// TwinCAT 3 PLC project sample_delivery
// ProgramVersion: 3.1.4023.0
// libraries:
//   LCLS Sample Delivery, * (SLAC - LCLS)
//   LCLS Vacuum, * (SLAC - LCLS)
//   Tc2_Standard, * (Beckhoff Automation GmbH)
//   Tc2_System, * (Beckhoff Automation GmbH)
//   Tc3_Module, * (Beckhoff Automation GmbH)
// project tree:
//   GVLs/ GVL_RCC.TcGVL, GVL_SDS.TcGVL
//   / PlcTask.TcTTO (not stored), SerialComm.TcTTO (not stored)
//   POUs/ MAIN.TcPOU, PRG_RCC.TcPOU, SerialTxRx.TcPOU (not stored)
// real-time tasks:
//   TASK PlcTask: cycle T#10ms, priority 20, ADS port 351
//   TASK SerialComm: cycle T#5ms, priority 1, ADS port 350
// I/O:
//   DEVICE MAIN (EtherCAT), AmsNetId 0.0.0.0.2.1
//     Term 65 (EK1200)
//     Box 23 (EP9128-0021)
//     Box 31 (EP9128-0021) [EP9128-0021 8x EtherCAT junction]
//       Term 73 (EP9128-1021) [EP9128-1021 8x EtherCAT junction - Dev A]
//       Term 74 (EP9128-2021) [EP9128-2021 8x EtherCAT junction - Dev B]
//     Box 75 (EP9128-0021) [EP9128-0021 8x EtherCAT junction]
//       Term 76 (EP9128-1021) [EP9128-1021 8x EtherCAT junction - Dev A]
//       Term 77 (EP9128-2021) [EP9128-2021 8x EtherCAT junction - Dev B]
//     Box 93 (EP9128-0021) [EP9128-0021 8x EtherCAT junction]
//       FEL-SIM [EP9128-0021 8x EtherCAT junction]
//         RCC [EK1100 EtherCAT Coupler (2A E-Bus)]
//           RCC-E1 (EL2004) [EL2004 4Ch. Dig. Output 24V, 0.5A]
//           RCC-E2 (EL1004) [EL1004 4Ch. Dig. Input 24V, 3ms]
//           RCC-E3 (EL2004) [EL2004 4Ch. Dig. Output 24V, 0.5A]
//           RCC-E4 (EL2004) [EL2004 4Ch. Dig. Output 24V, 0.5A]
//           RCC-E5 (EL1004) [EL1004 4Ch. Dig. Input 24V, 3ms]
//           RCC-E6 (EL3314) [EL3314 4Ch. Ana. Input Thermocouple (TC)]
//           RCC-E7 (EL3174) [EL3174 4Ch. Ana. Input +/-10V Diff., +/-20mA SingleEnded, 16 Bit]
//           RCC-E8 (EL9011) [EL9011 End Terminal]
//         Term 87 (EP9128-1021) [EP9128-1021 8x EtherCAT junction - Dev A]
//         Term 88 (EP9128-2021) [EP9128-2021 8x EtherCAT junction - Dev B]
//       FEL-SIM-RCC (EP2339-0021) [EP2339-0021 16 Ch. Dig. Input/Output 24V, 0,5A, M8]
//       FEL-SIM-PCM (EP4374-0002) [EP4374-0002 2Ch. Ana. Input +/-10V, 0-10V, 0/4-20mA configurable; 2Ch. Ana. Output +/-10V, 0-10V, 0/4-20mA configurable]
//       Term 94 (EP9128-1021) [EP9128-1021 8x EtherCAT junction - Dev A]
//       Term 95 (EP9128-2021) [EP9128-2021 8x EtherCAT junction - Dev B]
//     WALL-RCC (EP2338-0001) [EP2338-0001 8 Ch. Dig. Input/Output 24V, 0,5A, M8]
//     WALL-RCC-PCM (EP4374-0002) [EP4374-0002 2Ch. Ana. Input +/-10V, 0-10V, 0/4-20mA configurable; 2Ch. Ana. Output +/-10V, 0-10V, 0/4-20mA configurable]
//     ALI (EP1111)
//     ALI_X (EP7041-0002)
//     ALI_Y (EP7041-0002)
//     ALI_Z (EP7041-0002)
//     ALI_X_ENC (EP5101-0011)
//     ALI_Gauges (EP3174-0002)
//     ALI_PropValve (EP7041-0002)
//     ALI_Y_ENC (EP5101-0011)
//     ALI_DIO (EP2338-0001)
//     M3 Selector A (EP1111)
//     M3 Selector A Digital IO (EP2338-1001)
//     M3 Selector A Serial IO (EP6002-0002)
//     M3 Selector B (EP1111)
//     M3 Selector B Digital IO (EP2338-1001)
//     M3 Selector B Serial IO (EP6002-0002)
//     PCM A (EP1111)
//     PCM A (EP4374-0002)
//     PCM A (EP3174-0002)
//     PCM A (EP6002-0002)
//     PCM B (EP1111)
//     PCM B (EP4374-0002)
//     PCM B (EP3174-0002)
//     PCM B (EP6002-0002)
//     Gas_Mani (EP1111)
//     Gas_Mani_NeedleValve (EP4374-0002)
//     Gas_Mani_ValveCtrl (EP2338-0001)
//     Gas_Mani_ValveRbk (EP2338-0001)
//     M3 Selector C (EP1111)
//     M3 Selector C Digital IO (EP2338-1001)
//     M3 Selector C Serial IO (EP6002-0002)
//     M3 Selector D (EP1111)
//     M3 Selector D Digital IO (EP2338-1001)
//     M3 Selector D Serial IO (EP6002-0002)
//     PCM C (EP1111)
//     PCM C (EP4374-0002)
//     PCM C (EP3174-0002)
//     PCM C (EP6002-0002)
//     PCM D (EP1111)
//     PCM D (EP4374-0002)
//     PCM D (EP3174-0002)
//     PCM D (EP6002-0002)
//     Bronkhorst MFM A
//     Bronkhorst MFM B
//     Bronkhorst MFM C
//     Bronkhorst MFM D
//     Solenoid Pair A (EP1111)
//     Solenoid Pair A Digital IO (EP2338-0001)
//     SC5 [EP9128-0021 8x EtherCAT junction]
//       Box 26 (EP9128-1021) [EP9128-1021 8x EtherCAT junction - Dev A]
//       Box 27 (EP9128-2021) [EP9128-2021 8x EtherCAT junction - Dev B]
//         SC4
//     Sensirion Flow Meter A (EP1111) [EP1111-0000 ID-Switch]
//     Sensirion Flow Meter A Serial 01 (EP6002-0002) [EP6002-0002 Interface (RS232/422/485)]
//     Sensirion Flow Meter A Serial 02 (EP6002-0002) [EP6002-0002 Interface (RS232/422/485)]
// variable links:
//   sample_delivery Instance <-> MAIN (EtherCAT)/Box 93 (EP9128-0021)/FEL-SIM-PCM (EP4374-0002)
//     PlcTask Inputs/PRG_FEL_SIM.PCM_RCC.stPropAir1.i_iPressRB <-> AI Inputs Channel 1/Value
//     PlcTask Inputs/PRG_FEL_SIM.PCM_RCC.stPropAir2.i_iPressRB <-> AI Inputs Channel 2/Value
//     PlcTask Outputs/PRG_FEL_SIM.PCM_RCC.stPropAir1.q_iPressCt <-> AO Outputs Channel 3/Analog output
//     PlcTask Outputs/PRG_FEL_SIM.PCM_RCC.stPropAir2.q_iPressCt <-> AO Outputs Channel 4/Analog output
//   sample_delivery Instance <-> MAIN (EtherCAT)/Box 93 (EP9128-0021)/FEL-SIM-RCC (EP2339-0021)
//     PlcTask Inputs/GVL_FEL_SIM.FEL_SIM_VRC_01.i_xOpnLS <-> Channel 1/Input
//     PlcTask Inputs/GVL_FEL_SIM.FEL_SIM_VRC_02.i_xOpnLS <-> Channel 2/Input
//     PlcTask Inputs/GVL_FEL_SIM.FEL_SIM_VRC_03.i_xOpnLS <-> Channel 3/Input
//     PlcTask Inputs/GVL_FEL_SIM.FEL_SIM_VRC_04.i_xOpnLS <-> Channel 4/Input
//     PlcTask Inputs/GVL_FEL_SIM.FEL_SIM_VRC_05.i_xOpnLS <-> Channel 5/Input
//     PlcTask Inputs/GVL_FEL_SIM.FEL_SIM_VRC_06.i_xOpnLS <-> Channel 6/Input
//     PlcTask Inputs/GVL_FEL_SIM.FEL_SIM_VRC_07.i_xOpnLS <-> Channel 7/Input
//     PlcTask Inputs/GVL_FEL_SIM.FEL_SIM_VRC_08.i_xOpnLS <-> Channel 8/Input
//     PlcTask Inputs/GVL_FEL_SIM.FEL_SIM_VRC_09.i_xOpnLS <-> Channel 9/Input
//     PlcTask Inputs/GVL_FEL_SIM.FEL_SIM_VRC_10.i_xOpnLS <-> Channel 10/Input
//     PlcTask Inputs/GVL_FEL_SIM.FEL_SIM_VRC_11.i_xOpnLS <-> Channel 11/Input
//     PlcTask Inputs/GVL_FEL_SIM.FEL_SIM_VRC_12.i_xOpnLS <-> Channel 12/Input
//     PlcTask Outputs/GVL_FEL_SIM.FEL_SIM_VRC_01.q_xOPN_DO <-> Channel 17/Output
//     PlcTask Outputs/GVL_FEL_SIM.FEL_SIM_VRC_02.q_xOPN_DO <-> Channel 18/Output
//     PlcTask Outputs/GVL_FEL_SIM.FEL_SIM_VRC_03.q_xOPN_DO <-> Channel 19/Output
//     PlcTask Outputs/GVL_FEL_SIM.FEL_SIM_VRC_04.q_xOPN_DO <-> Channel 20/Output
//     PlcTask Outputs/GVL_FEL_SIM.FEL_SIM_VRC_05.q_xOPN_DO <-> Channel 21/Output
//     PlcTask Outputs/GVL_FEL_SIM.FEL_SIM_VRC_06.q_xOPN_DO <-> Channel 22/Output
//     PlcTask Outputs/GVL_FEL_SIM.FEL_SIM_VRC_07.q_xOPN_DO <-> Channel 23/Output
//     PlcTask Outputs/GVL_FEL_SIM.FEL_SIM_VRC_08.q_xOPN_DO <-> Channel 24/Output
//     PlcTask Outputs/GVL_FEL_SIM.FEL_SIM_VRC_09.q_xOPN_DO <-> Channel 25/Output
//     PlcTask Outputs/GVL_FEL_SIM.FEL_SIM_VRC_10.q_xOPN_DO <-> Channel 26/Output
//     PlcTask Outputs/GVL_FEL_SIM.FEL_SIM_VRC_11.q_xOPN_DO <-> Channel 27/Output
//     PlcTask Outputs/GVL_FEL_SIM.FEL_SIM_VRC_12.q_xOPN_DO <-> Channel 28/Output
//   sample_delivery Instance <-> MAIN (EtherCAT)/Box 93 (EP9128-0021)/FEL-SIM/RCC/RCC-E6 (EL3314)
//     PlcTask Inputs/GVL_Recirculation.RCC_STC_01.bError <-> TC Inputs Channel 1/Status/Error
//     PlcTask Inputs/GVL_Recirculation.RCC_STC_01.bOverrange <-> TC Inputs Channel 1/Status/Overrange
//     PlcTask Inputs/GVL_Recirculation.RCC_STC_01.bUnderrange <-> TC Inputs Channel 1/Status/Underrange
//     PlcTask Inputs/GVL_Recirculation.RCC_STC_01.iRaw <-> TC Inputs Channel 1/Value
//   sample_delivery Instance <-> MAIN (EtherCAT)/Box 93 (EP9128-0021)/FEL-SIM/RCC/RCC-E7 (EL3174)
//     PlcTask Inputs/GVL_Recirculation.RCC_GCP_01.i_iPRESS_R <-> AI Standard Channel 1/Value
//   sample_delivery Instance <-> MAIN (EtherCAT)/Bronkhorst MFM A
//     PlcTask Inputs/GVL_SDS.BronkhorstA.stMFM.i_rFlow <-> TxPDO Map/fMeasure
//     PlcTask Outputs/GVL_SDS.BronkhorstA.stMFM.q_rSetpoint <-> RxPDO Map/fSetpoint
//   sample_delivery Instance <-> MAIN (EtherCAT)/Bronkhorst MFM B
//     PlcTask Inputs/GVL_SDS.BronkhorstB.stMFM.i_rFlow <-> TxPDO Map/fMeasure
//     PlcTask Outputs/GVL_SDS.BronkhorstB.stMFM.q_rSetpoint <-> RxPDO Map/fSetpoint
//   sample_delivery Instance <-> MAIN (EtherCAT)/Bronkhorst MFM C
//     PlcTask Inputs/GVL_SDS.BronkhorstC.stMFM.i_rFlow <-> TxPDO Map/fMeasure
//     PlcTask Outputs/GVL_SDS.BronkhorstC.stMFM.q_rSetpoint <-> RxPDO Map/fSetpoint
//   sample_delivery Instance <-> MAIN (EtherCAT)/Bronkhorst MFM D
//     PlcTask Inputs/GVL_SDS.BronkhorstD.stMFM.i_rFlow <-> TxPDO Map/fMeasure
//     PlcTask Outputs/GVL_SDS.BronkhorstD.stMFM.q_rSetpoint <-> RxPDO Map/fSetpoint
//   sample_delivery Instance <-> MAIN (EtherCAT)/Gas_Mani (EP1111)
//     PlcTask Inputs/GVL_SDS.GasMan.stBaseIO.i_SyncUnitWC <-> WcState/WcState
//   sample_delivery Instance <-> MAIN (EtherCAT)/Gas_Mani_ValveCtrl (EP2338-0001)
//     PlcTask Outputs/GVL_SDS.GasMan.stValve[{1..7}].qxDO <-> Channel {9..15}/Output  (7 links)
//   sample_delivery Instance <-> MAIN (EtherCAT)/Gas_Mani_ValveRbk (EP2338-0001)
//     PlcTask Inputs/GVL_SDS.GasMan.stValve[{1..7}].ixOPN <-> Channel {1..7}/Input  (7 links)
//   sample_delivery Instance <-> MAIN (EtherCAT)/M3 Selector A (EP1111)
//     PlcTask Inputs/GVL_SDS.M3SelectorA.stBaseIO.i_SyncUnitWC <-> WcState/WcState
//   sample_delivery Instance <-> MAIN (EtherCAT)/M3 Selector A Digital IO (EP2338-1001)
//     PlcTask Outputs/GVL_SDS.M3SelectorA.stShaker01.q_xPwrDO <-> Channel 9/Output
//     PlcTask Outputs/GVL_SDS.M3SelectorA.stShaker02.q_xPwrDO <-> Channel 10/Output
//     PlcTask Outputs/GVL_SDS.M3SelectorA.stShaker03.q_xPwrDO <-> Channel 11/Output
//     PlcTask Outputs/GVL_SDS.M3SelectorA.stShaker04.q_xPwrDO <-> Channel 12/Output
//   sample_delivery Instance <-> MAIN (EtherCAT)/M3 Selector A Serial IO (EP6002-0002)
//     SerialComm Inputs/GVL_SDS.M3SelectorA.stSensSerial.stComIn/D <-> COM TxPDO-Map Inputs Channel 1/Data In 0
//     SerialComm Inputs/GVL_SDS.M3SelectorA.stSensSerial.stComIn/D @bit {8..168 step 8} <-> COM TxPDO-Map Inputs Channel 1/Data In {1..21}  (21 links)
//     SerialComm Inputs/GVL_SDS.M3SelectorA.stSensSerial.stComIn/Status <-> COM TxPDO-Map Inputs Channel 1/Status
//     SerialComm Inputs/GVL_SDS.M3SelectorA.stViciSerial.stComIn/D <-> COM TxPDO-Map Inputs Channel 2/Data In 0
//     SerialComm Inputs/GVL_SDS.M3SelectorA.stViciSerial.stComIn/D @bit {8..168 step 8} <-> COM TxPDO-Map Inputs Channel 2/Data In {1..21}  (21 links)
//     SerialComm Inputs/GVL_SDS.M3SelectorA.stViciSerial.stComIn/Status <-> COM TxPDO-Map Inputs Channel 2/Status
//     SerialComm Outputs/GVL_SDS.M3SelectorA.stSensSerial.stComOut/Ctrl <-> COM RxPDO-Map Outputs Channel 1/Ctrl
//     SerialComm Outputs/GVL_SDS.M3SelectorA.stSensSerial.stComOut/D <-> COM RxPDO-Map Outputs Channel 1/Data Out 0
//     SerialComm Outputs/GVL_SDS.M3SelectorA.stSensSerial.stComOut/D @bit {8..168 step 8} <-> COM RxPDO-Map Outputs Channel 1/Data Out {1..21}  (21 links)
//     SerialComm Outputs/GVL_SDS.M3SelectorA.stViciSerial.stComOut/Ctrl <-> COM RxPDO-Map Outputs Channel 2/Ctrl
//     SerialComm Outputs/GVL_SDS.M3SelectorA.stViciSerial.stComOut/D <-> COM RxPDO-Map Outputs Channel 2/Data Out 0
//     SerialComm Outputs/GVL_SDS.M3SelectorA.stViciSerial.stComOut/D @bit {8..168 step 8} <-> COM RxPDO-Map Outputs Channel 2/Data Out {1..21}  (21 links)
//   sample_delivery Instance <-> MAIN (EtherCAT)/M3 Selector B (EP1111)
//     PlcTask Inputs/GVL_SDS.M3SelectorB.stBaseIO.i_SyncUnitWC <-> WcState/WcState
//   sample_delivery Instance <-> MAIN (EtherCAT)/M3 Selector B Digital IO (EP2338-1001)
//     PlcTask Outputs/GVL_SDS.M3SelectorB.stShaker01.q_xPwrDO <-> Channel 9/Output
//     PlcTask Outputs/GVL_SDS.M3SelectorB.stShaker02.q_xPwrDO <-> Channel 10/Output
//     PlcTask Outputs/GVL_SDS.M3SelectorB.stShaker03.q_xPwrDO <-> Channel 11/Output
//     PlcTask Outputs/GVL_SDS.M3SelectorB.stShaker04.q_xPwrDO <-> Channel 12/Output
//   sample_delivery Instance <-> MAIN (EtherCAT)/M3 Selector B Serial IO (EP6002-0002)
//     SerialComm Inputs/GVL_SDS.M3SelectorB.stSensSerial.stComIn/D <-> COM TxPDO-Map Inputs Channel 1/Data In 0
//     SerialComm Inputs/GVL_SDS.M3SelectorB.stSensSerial.stComIn/D @bit {8..168 step 8} <-> COM TxPDO-Map Inputs Channel 1/Data In {1..21}  (21 links)
//     SerialComm Inputs/GVL_SDS.M3SelectorB.stSensSerial.stComIn/Status <-> COM TxPDO-Map Inputs Channel 1/Status
//     SerialComm Inputs/GVL_SDS.M3SelectorB.stViciSerial.stComIn/D <-> COM TxPDO-Map Inputs Channel 2/Data In 0
//     SerialComm Inputs/GVL_SDS.M3SelectorB.stViciSerial.stComIn/D @bit {8..168 step 8} <-> COM TxPDO-Map Inputs Channel 2/Data In {1..21}  (21 links)
//     SerialComm Inputs/GVL_SDS.M3SelectorB.stViciSerial.stComIn/Status <-> COM TxPDO-Map Inputs Channel 2/Status
//     SerialComm Outputs/GVL_SDS.M3SelectorB.stSensSerial.stComOut/Ctrl <-> COM RxPDO-Map Outputs Channel 1/Ctrl
//     SerialComm Outputs/GVL_SDS.M3SelectorB.stSensSerial.stComOut/D <-> COM RxPDO-Map Outputs Channel 1/Data Out 0
//     SerialComm Outputs/GVL_SDS.M3SelectorB.stSensSerial.stComOut/D @bit {8..168 step 8} <-> COM RxPDO-Map Outputs Channel 1/Data Out {1..21}  (21 links)
//     SerialComm Outputs/GVL_SDS.M3SelectorB.stViciSerial.stComOut/Ctrl <-> COM RxPDO-Map Outputs Channel 2/Ctrl
//     SerialComm Outputs/GVL_SDS.M3SelectorB.stViciSerial.stComOut/D <-> COM RxPDO-Map Outputs Channel 2/Data Out 0
//     SerialComm Outputs/GVL_SDS.M3SelectorB.stViciSerial.stComOut/D @bit {8..168 step 8} <-> COM RxPDO-Map Outputs Channel 2/Data Out {1..21}  (21 links)
//   sample_delivery Instance <-> MAIN (EtherCAT)/M3 Selector C (EP1111)
//     PlcTask Inputs/GVL_SDS.M3SelectorC.stBaseIO.i_SyncUnitWC <-> WcState/WcState
//   sample_delivery Instance <-> MAIN (EtherCAT)/M3 Selector C Digital IO (EP2338-1001)
//     PlcTask Outputs/GVL_SDS.M3SelectorC.stShaker01.q_xPwrDO <-> Channel 9/Output
//     PlcTask Outputs/GVL_SDS.M3SelectorC.stShaker02.q_xPwrDO <-> Channel 10/Output
//     PlcTask Outputs/GVL_SDS.M3SelectorC.stShaker03.q_xPwrDO <-> Channel 11/Output
//     PlcTask Outputs/GVL_SDS.M3SelectorC.stShaker04.q_xPwrDO <-> Channel 12/Output
//   sample_delivery Instance <-> MAIN (EtherCAT)/M3 Selector C Serial IO (EP6002-0002)
//     SerialComm Inputs/GVL_SDS.M3SelectorC.stSensSerial.stComIn/D <-> COM TxPDO-Map Inputs Channel 1/Data In 0
//     SerialComm Inputs/GVL_SDS.M3SelectorC.stSensSerial.stComIn/D @bit {8..168 step 8} <-> COM TxPDO-Map Inputs Channel 1/Data In {1..21}  (21 links)
//     SerialComm Inputs/GVL_SDS.M3SelectorC.stSensSerial.stComIn/Status <-> COM TxPDO-Map Inputs Channel 1/Status
//     SerialComm Inputs/GVL_SDS.M3SelectorC.stViciSerial.stComIn/D <-> COM TxPDO-Map Inputs Channel 2/Data In 0
//     SerialComm Inputs/GVL_SDS.M3SelectorC.stViciSerial.stComIn/D @bit {8..168 step 8} <-> COM TxPDO-Map Inputs Channel 2/Data In {1..21}  (21 links)
//     SerialComm Inputs/GVL_SDS.M3SelectorC.stViciSerial.stComIn/Status <-> COM TxPDO-Map Inputs Channel 2/Status
//     SerialComm Outputs/GVL_SDS.M3SelectorC.stSensSerial.stComOut/Ctrl <-> COM RxPDO-Map Outputs Channel 1/Ctrl
//     SerialComm Outputs/GVL_SDS.M3SelectorC.stSensSerial.stComOut/D <-> COM RxPDO-Map Outputs Channel 1/Data Out 0
//     SerialComm Outputs/GVL_SDS.M3SelectorC.stSensSerial.stComOut/D @bit {8..168 step 8} <-> COM RxPDO-Map Outputs Channel 1/Data Out {1..21}  (21 links)
//     SerialComm Outputs/GVL_SDS.M3SelectorC.stViciSerial.stComOut/Ctrl <-> COM RxPDO-Map Outputs Channel 2/Ctrl
//     SerialComm Outputs/GVL_SDS.M3SelectorC.stViciSerial.stComOut/D <-> COM RxPDO-Map Outputs Channel 2/Data Out 0
//     SerialComm Outputs/GVL_SDS.M3SelectorC.stViciSerial.stComOut/D @bit {8..168 step 8} <-> COM RxPDO-Map Outputs Channel 2/Data Out {1..21}  (21 links)
//   sample_delivery Instance <-> MAIN (EtherCAT)/M3 Selector D (EP1111)
//     PlcTask Inputs/GVL_SDS.M3SelectorD.stBaseIO.i_SyncUnitWC <-> WcState/WcState
//   sample_delivery Instance <-> MAIN (EtherCAT)/M3 Selector D Digital IO (EP2338-1001)
//     PlcTask Outputs/GVL_SDS.M3SelectorD.stShaker01.q_xPwrDO <-> Channel 9/Output
//     PlcTask Outputs/GVL_SDS.M3SelectorD.stShaker02.q_xPwrDO <-> Channel 10/Output
//     PlcTask Outputs/GVL_SDS.M3SelectorD.stShaker03.q_xPwrDO <-> Channel 11/Output
//     PlcTask Outputs/GVL_SDS.M3SelectorD.stShaker04.q_xPwrDO <-> Channel 12/Output
//   sample_delivery Instance <-> MAIN (EtherCAT)/M3 Selector D Serial IO (EP6002-0002)
//     SerialComm Inputs/GVL_SDS.M3SelectorD.stSensSerial.stComIn/D <-> COM TxPDO-Map Inputs Channel 1/Data In 0
//     SerialComm Inputs/GVL_SDS.M3SelectorD.stSensSerial.stComIn/D @bit {8..168 step 8} <-> COM TxPDO-Map Inputs Channel 1/Data In {1..21}  (21 links)
//     SerialComm Inputs/GVL_SDS.M3SelectorD.stSensSerial.stComIn/Status <-> COM TxPDO-Map Inputs Channel 1/Status
//     SerialComm Inputs/GVL_SDS.M3SelectorD.stViciSerial.stComIn/D <-> COM TxPDO-Map Inputs Channel 2/Data In 0
//     SerialComm Inputs/GVL_SDS.M3SelectorD.stViciSerial.stComIn/D @bit {8..168 step 8} <-> COM TxPDO-Map Inputs Channel 2/Data In {1..21}  (21 links)
//     SerialComm Inputs/GVL_SDS.M3SelectorD.stViciSerial.stComIn/Status <-> COM TxPDO-Map Inputs Channel 2/Status
//     SerialComm Outputs/GVL_SDS.M3SelectorD.stSensSerial.stComOut/Ctrl <-> COM RxPDO-Map Outputs Channel 1/Ctrl
//     SerialComm Outputs/GVL_SDS.M3SelectorD.stSensSerial.stComOut/D <-> COM RxPDO-Map Outputs Channel 1/Data Out 0
//     SerialComm Outputs/GVL_SDS.M3SelectorD.stSensSerial.stComOut/D @bit {8..168 step 8} <-> COM RxPDO-Map Outputs Channel 1/Data Out {1..21}  (21 links)
//     SerialComm Outputs/GVL_SDS.M3SelectorD.stViciSerial.stComOut/Ctrl <-> COM RxPDO-Map Outputs Channel 2/Ctrl
//     SerialComm Outputs/GVL_SDS.M3SelectorD.stViciSerial.stComOut/D <-> COM RxPDO-Map Outputs Channel 2/Data Out 0
//     SerialComm Outputs/GVL_SDS.M3SelectorD.stViciSerial.stComOut/D @bit {8..168 step 8} <-> COM RxPDO-Map Outputs Channel 2/Data Out {1..21}  (21 links)
//   sample_delivery Instance <-> MAIN (EtherCAT)/PCM A (EP1111)
//     PlcTask Inputs/GVL_SDS.PCMA.stBaseIO.i_SyncUnitWC <-> WcState/WcState
//   sample_delivery Instance <-> MAIN (EtherCAT)/PCM A (EP4374-0002)
//     PlcTask Inputs/GVL_SDS.PCMA.stPropAir1.i_iPressRB <-> AI Inputs Channel 1/Value
//     PlcTask Inputs/GVL_SDS.PCMA.stPropAir2.i_iPressRB <-> AI Inputs Channel 2/Value
//     PlcTask Outputs/GVL_SDS.PCMA.stPropAir1.q_iPressCt <-> AO Outputs Channel 3/Analog output
//     PlcTask Outputs/GVL_SDS.PCMA.stPropAir2.q_iPressCt <-> AO Outputs Channel 4/Analog output
//   sample_delivery Instance <-> MAIN (EtherCAT)/PCM A (EP6002-0002)
//     SerialComm Inputs/GVL_SDS.PCMA.stSerial1.stComIn/D <-> COM TxPDO-Map Inputs Channel 1/Data In 0
//     SerialComm Inputs/GVL_SDS.PCMA.stSerial2.stComIn/D <-> COM TxPDO-Map Inputs Channel 2/Data In 0
//     SerialComm Inputs/GVL_SDS.PCMA.stSerial1.stComIn/D @bit 8 <-> COM TxPDO-Map Inputs Channel 1/Data In 1
//     SerialComm Inputs/GVL_SDS.PCMA.stSerial1.stComIn/D @bit 80 <-> COM TxPDO-Map Inputs Channel 1/Data In 10
//     SerialComm Inputs/GVL_SDS.PCMA.stSerial1.stComIn/D @bit 88 <-> COM TxPDO-Map Inputs Channel 1/Data In 11
//     SerialComm Inputs/GVL_SDS.PCMA.stSerial1.stComIn/D @bit 96 <-> COM TxPDO-Map Inputs Channel 1/Data In 12
//     SerialComm Inputs/GVL_SDS.PCMA.stSerial1.stComIn/D @bit 104 <-> COM TxPDO-Map Inputs Channel 1/Data In 13
//     SerialComm Inputs/GVL_SDS.PCMA.stSerial1.stComIn/D @bit 112 <-> COM TxPDO-Map Inputs Channel 1/Data In 14
//     SerialComm Inputs/GVL_SDS.PCMA.stSerial1.stComIn/D @bit 120 <-> COM TxPDO-Map Inputs Channel 1/Data In 15
//     SerialComm Inputs/GVL_SDS.PCMA.stSerial1.stComIn/D @bit 128 <-> COM TxPDO-Map Inputs Channel 1/Data In 16
//     SerialComm Inputs/GVL_SDS.PCMA.stSerial1.stComIn/D @bit 136 <-> COM TxPDO-Map Inputs Channel 1/Data In 17
//     SerialComm Inputs/GVL_SDS.PCMA.stSerial1.stComIn/D @bit 144 <-> COM TxPDO-Map Inputs Channel 1/Data In 18
//     SerialComm Inputs/GVL_SDS.PCMA.stSerial1.stComIn/D @bit 152 <-> COM TxPDO-Map Inputs Channel 1/Data In 19
//     SerialComm Inputs/GVL_SDS.PCMA.stSerial1.stComIn/D @bit 16 <-> COM TxPDO-Map Inputs Channel 1/Data In 2
//     SerialComm Inputs/GVL_SDS.PCMA.stSerial1.stComIn/D @bit 160 <-> COM TxPDO-Map Inputs Channel 1/Data In 20
//     SerialComm Inputs/GVL_SDS.PCMA.stSerial1.stComIn/D @bit 168 <-> COM TxPDO-Map Inputs Channel 1/Data In 21
//     SerialComm Inputs/GVL_SDS.PCMA.stSerial1.stComIn/D @bit 24 <-> COM TxPDO-Map Inputs Channel 1/Data In 3
//     SerialComm Inputs/GVL_SDS.PCMA.stSerial1.stComIn/D @bit 32 <-> COM TxPDO-Map Inputs Channel 1/Data In 4
//     SerialComm Inputs/GVL_SDS.PCMA.stSerial1.stComIn/D @bit 40 <-> COM TxPDO-Map Inputs Channel 1/Data In 5
//     SerialComm Inputs/GVL_SDS.PCMA.stSerial1.stComIn/D @bit 48 <-> COM TxPDO-Map Inputs Channel 1/Data In 6
//     SerialComm Inputs/GVL_SDS.PCMA.stSerial1.stComIn/D @bit 56 <-> COM TxPDO-Map Inputs Channel 1/Data In 7
//     SerialComm Inputs/GVL_SDS.PCMA.stSerial1.stComIn/D @bit 64 <-> COM TxPDO-Map Inputs Channel 1/Data In 8
//     SerialComm Inputs/GVL_SDS.PCMA.stSerial1.stComIn/D @bit 72 <-> COM TxPDO-Map Inputs Channel 1/Data In 9
//     SerialComm Inputs/GVL_SDS.PCMA.stSerial2.stComIn/D @bit 8 <-> COM TxPDO-Map Inputs Channel 2/Data In 1
//     SerialComm Inputs/GVL_SDS.PCMA.stSerial2.stComIn/D @bit 80 <-> COM TxPDO-Map Inputs Channel 2/Data In 10
//     SerialComm Inputs/GVL_SDS.PCMA.stSerial2.stComIn/D @bit 88 <-> COM TxPDO-Map Inputs Channel 2/Data In 11
//     SerialComm Inputs/GVL_SDS.PCMA.stSerial2.stComIn/D @bit 96 <-> COM TxPDO-Map Inputs Channel 2/Data In 12
//     SerialComm Inputs/GVL_SDS.PCMA.stSerial2.stComIn/D @bit 104 <-> COM TxPDO-Map Inputs Channel 2/Data In 13
//     SerialComm Inputs/GVL_SDS.PCMA.stSerial2.stComIn/D @bit 112 <-> COM TxPDO-Map Inputs Channel 2/Data In 14
//     SerialComm Inputs/GVL_SDS.PCMA.stSerial2.stComIn/D @bit 120 <-> COM TxPDO-Map Inputs Channel 2/Data In 15
//     SerialComm Inputs/GVL_SDS.PCMA.stSerial2.stComIn/D @bit 128 <-> COM TxPDO-Map Inputs Channel 2/Data In 16
//     SerialComm Inputs/GVL_SDS.PCMA.stSerial2.stComIn/D @bit 136 <-> COM TxPDO-Map Inputs Channel 2/Data In 17
//     SerialComm Inputs/GVL_SDS.PCMA.stSerial2.stComIn/D @bit 144 <-> COM TxPDO-Map Inputs Channel 2/Data In 18
//     SerialComm Inputs/GVL_SDS.PCMA.stSerial2.stComIn/D @bit 152 <-> COM TxPDO-Map Inputs Channel 2/Data In 19
//     SerialComm Inputs/GVL_SDS.PCMA.stSerial2.stComIn/D @bit 16 <-> COM TxPDO-Map Inputs Channel 2/Data In 2
//     SerialComm Inputs/GVL_SDS.PCMA.stSerial2.stComIn/D @bit 160 <-> COM TxPDO-Map Inputs Channel 2/Data In 20
//     SerialComm Inputs/GVL_SDS.PCMA.stSerial2.stComIn/D @bit 168 <-> COM TxPDO-Map Inputs Channel 2/Data In 21
//     SerialComm Inputs/GVL_SDS.PCMA.stSerial2.stComIn/D @bit 24 <-> COM TxPDO-Map Inputs Channel 2/Data In 3
//     SerialComm Inputs/GVL_SDS.PCMA.stSerial2.stComIn/D @bit 32 <-> COM TxPDO-Map Inputs Channel 2/Data In 4
//     SerialComm Inputs/GVL_SDS.PCMA.stSerial2.stComIn/D @bit 40 <-> COM TxPDO-Map Inputs Channel 2/Data In 5
//     SerialComm Inputs/GVL_SDS.PCMA.stSerial2.stComIn/D @bit 48 <-> COM TxPDO-Map Inputs Channel 2/Data In 6
//     SerialComm Inputs/GVL_SDS.PCMA.stSerial2.stComIn/D @bit 56 <-> COM TxPDO-Map Inputs Channel 2/Data In 7
//     SerialComm Inputs/GVL_SDS.PCMA.stSerial2.stComIn/D @bit 64 <-> COM TxPDO-Map Inputs Channel 2/Data In 8
//     SerialComm Inputs/GVL_SDS.PCMA.stSerial2.stComIn/D @bit 72 <-> COM TxPDO-Map Inputs Channel 2/Data In 9
//     SerialComm Inputs/GVL_SDS.PCMA.stSerial1.stComIn/Status <-> COM TxPDO-Map Inputs Channel 1/Status
//     SerialComm Inputs/GVL_SDS.PCMA.stSerial2.stComIn/Status <-> COM TxPDO-Map Inputs Channel 2/Status
//     SerialComm Outputs/GVL_SDS.PCMA.stSerial1.stComOut/Ctrl <-> COM RxPDO-Map Outputs Channel 1/Ctrl
//     SerialComm Outputs/GVL_SDS.PCMA.stSerial2.stComOut/Ctrl <-> COM RxPDO-Map Outputs Channel 2/Ctrl
//     SerialComm Outputs/GVL_SDS.PCMA.stSerial1.stComOut/D <-> COM RxPDO-Map Outputs Channel 1/Data Out 0
//     SerialComm Outputs/GVL_SDS.PCMA.stSerial2.stComOut/D <-> COM RxPDO-Map Outputs Channel 2/Data Out 0
//     SerialComm Outputs/GVL_SDS.PCMA.stSerial1.stComOut/D @bit 8 <-> COM RxPDO-Map Outputs Channel 1/Data Out 1
//     SerialComm Outputs/GVL_SDS.PCMA.stSerial1.stComOut/D @bit 80 <-> COM RxPDO-Map Outputs Channel 1/Data Out 10
//     SerialComm Outputs/GVL_SDS.PCMA.stSerial1.stComOut/D @bit 88 <-> COM RxPDO-Map Outputs Channel 1/Data Out 11
//     SerialComm Outputs/GVL_SDS.PCMA.stSerial1.stComOut/D @bit 96 <-> COM RxPDO-Map Outputs Channel 1/Data Out 12
//     SerialComm Outputs/GVL_SDS.PCMA.stSerial1.stComOut/D @bit 104 <-> COM RxPDO-Map Outputs Channel 1/Data Out 13
//     SerialComm Outputs/GVL_SDS.PCMA.stSerial1.stComOut/D @bit 112 <-> COM RxPDO-Map Outputs Channel 1/Data Out 14
//     SerialComm Outputs/GVL_SDS.PCMA.stSerial1.stComOut/D @bit 120 <-> COM RxPDO-Map Outputs Channel 1/Data Out 15
//     SerialComm Outputs/GVL_SDS.PCMA.stSerial1.stComOut/D @bit 128 <-> COM RxPDO-Map Outputs Channel 1/Data Out 16
//     SerialComm Outputs/GVL_SDS.PCMA.stSerial1.stComOut/D @bit 136 <-> COM RxPDO-Map Outputs Channel 1/Data Out 17
//     SerialComm Outputs/GVL_SDS.PCMA.stSerial1.stComOut/D @bit 144 <-> COM RxPDO-Map Outputs Channel 1/Data Out 18
//     SerialComm Outputs/GVL_SDS.PCMA.stSerial1.stComOut/D @bit 152 <-> COM RxPDO-Map Outputs Channel 1/Data Out 19
//     SerialComm Outputs/GVL_SDS.PCMA.stSerial1.stComOut/D @bit 16 <-> COM RxPDO-Map Outputs Channel 1/Data Out 2
//     SerialComm Outputs/GVL_SDS.PCMA.stSerial1.stComOut/D @bit 160 <-> COM RxPDO-Map Outputs Channel 1/Data Out 20
//     SerialComm Outputs/GVL_SDS.PCMA.stSerial1.stComOut/D @bit 168 <-> COM RxPDO-Map Outputs Channel 1/Data Out 21
//     SerialComm Outputs/GVL_SDS.PCMA.stSerial1.stComOut/D @bit 24 <-> COM RxPDO-Map Outputs Channel 1/Data Out 3
//     SerialComm Outputs/GVL_SDS.PCMA.stSerial1.stComOut/D @bit 32 <-> COM RxPDO-Map Outputs Channel 1/Data Out 4
//     SerialComm Outputs/GVL_SDS.PCMA.stSerial1.stComOut/D @bit 40 <-> COM RxPDO-Map Outputs Channel 1/Data Out 5
//     SerialComm Outputs/GVL_SDS.PCMA.stSerial1.stComOut/D @bit 48 <-> COM RxPDO-Map Outputs Channel 1/Data Out 6
//     SerialComm Outputs/GVL_SDS.PCMA.stSerial1.stComOut/D @bit 56 <-> COM RxPDO-Map Outputs Channel 1/Data Out 7
//     SerialComm Outputs/GVL_SDS.PCMA.stSerial1.stComOut/D @bit 64 <-> COM RxPDO-Map Outputs Channel 1/Data Out 8
//     SerialComm Outputs/GVL_SDS.PCMA.stSerial1.stComOut/D @bit 72 <-> COM RxPDO-Map Outputs Channel 1/Data Out 9
//     SerialComm Outputs/GVL_SDS.PCMA.stSerial2.stComOut/D @bit 8 <-> COM RxPDO-Map Outputs Channel 2/Data Out 1
//     SerialComm Outputs/GVL_SDS.PCMA.stSerial2.stComOut/D @bit 80 <-> COM RxPDO-Map Outputs Channel 2/Data Out 10
//     SerialComm Outputs/GVL_SDS.PCMA.stSerial2.stComOut/D @bit 88 <-> COM RxPDO-Map Outputs Channel 2/Data Out 11
//     SerialComm Outputs/GVL_SDS.PCMA.stSerial2.stComOut/D @bit 96 <-> COM RxPDO-Map Outputs Channel 2/Data Out 12
//     SerialComm Outputs/GVL_SDS.PCMA.stSerial2.stComOut/D @bit 104 <-> COM RxPDO-Map Outputs Channel 2/Data Out 13
//     SerialComm Outputs/GVL_SDS.PCMA.stSerial2.stComOut/D @bit 112 <-> COM RxPDO-Map Outputs Channel 2/Data Out 14
//     SerialComm Outputs/GVL_SDS.PCMA.stSerial2.stComOut/D @bit 120 <-> COM RxPDO-Map Outputs Channel 2/Data Out 15
//     SerialComm Outputs/GVL_SDS.PCMA.stSerial2.stComOut/D @bit 128 <-> COM RxPDO-Map Outputs Channel 2/Data Out 16
//     SerialComm Outputs/GVL_SDS.PCMA.stSerial2.stComOut/D @bit 136 <-> COM RxPDO-Map Outputs Channel 2/Data Out 17
//     SerialComm Outputs/GVL_SDS.PCMA.stSerial2.stComOut/D @bit 144 <-> COM RxPDO-Map Outputs Channel 2/Data Out 18
//     SerialComm Outputs/GVL_SDS.PCMA.stSerial2.stComOut/D @bit 152 <-> COM RxPDO-Map Outputs Channel 2/Data Out 19
//     SerialComm Outputs/GVL_SDS.PCMA.stSerial2.stComOut/D @bit 16 <-> COM RxPDO-Map Outputs Channel 2/Data Out 2
//     SerialComm Outputs/GVL_SDS.PCMA.stSerial2.stComOut/D @bit 160 <-> COM RxPDO-Map Outputs Channel 2/Data Out 20
//     SerialComm Outputs/GVL_SDS.PCMA.stSerial2.stComOut/D @bit 168 <-> COM RxPDO-Map Outputs Channel 2/Data Out 21
//     SerialComm Outputs/GVL_SDS.PCMA.stSerial2.stComOut/D @bit 24 <-> COM RxPDO-Map Outputs Channel 2/Data Out 3
//     SerialComm Outputs/GVL_SDS.PCMA.stSerial2.stComOut/D @bit 32 <-> COM RxPDO-Map Outputs Channel 2/Data Out 4
//     SerialComm Outputs/GVL_SDS.PCMA.stSerial2.stComOut/D @bit 40 <-> COM RxPDO-Map Outputs Channel 2/Data Out 5
//     SerialComm Outputs/GVL_SDS.PCMA.stSerial2.stComOut/D @bit 48 <-> COM RxPDO-Map Outputs Channel 2/Data Out 6
//     SerialComm Outputs/GVL_SDS.PCMA.stSerial2.stComOut/D @bit 56 <-> COM RxPDO-Map Outputs Channel 2/Data Out 7
//     SerialComm Outputs/GVL_SDS.PCMA.stSerial2.stComOut/D @bit 64 <-> COM RxPDO-Map Outputs Channel 2/Data Out 8
//     SerialComm Outputs/GVL_SDS.PCMA.stSerial2.stComOut/D @bit 72 <-> COM RxPDO-Map Outputs Channel 2/Data Out 9
//   sample_delivery Instance <-> MAIN (EtherCAT)/PCM B (EP1111)
//     PlcTask Inputs/GVL_SDS.PCMB.stBaseIO.i_SyncUnitWC <-> WcState/WcState
//   sample_delivery Instance <-> MAIN (EtherCAT)/PCM B (EP4374-0002)
//     PlcTask Inputs/GVL_SDS.PCMB.stPropAir1.i_iPressRB <-> AI Inputs Channel 1/Value
//     PlcTask Inputs/GVL_SDS.PCMB.stPropAir2.i_iPressRB <-> AI Inputs Channel 2/Value
//     PlcTask Outputs/GVL_SDS.PCMB.stPropAir1.q_iPressCt <-> AO Outputs Channel 3/Analog output
//     PlcTask Outputs/GVL_SDS.PCMB.stPropAir2.q_iPressCt <-> AO Outputs Channel 4/Analog output
//   sample_delivery Instance <-> MAIN (EtherCAT)/PCM B (EP6002-0002)
//     SerialComm Inputs/GVL_SDS.PCMB.stSerial1.stComIn/D <-> COM TxPDO-Map Inputs Channel 1/Data In 0
//     SerialComm Inputs/GVL_SDS.PCMB.stSerial2.stComIn/D <-> COM TxPDO-Map Inputs Channel 2/Data In 0
//     SerialComm Inputs/GVL_SDS.PCMB.stSerial1.stComIn/D @bit 8 <-> COM TxPDO-Map Inputs Channel 1/Data In 1
//     SerialComm Inputs/GVL_SDS.PCMB.stSerial1.stComIn/D @bit 80 <-> COM TxPDO-Map Inputs Channel 1/Data In 10
//     SerialComm Inputs/GVL_SDS.PCMB.stSerial1.stComIn/D @bit 88 <-> COM TxPDO-Map Inputs Channel 1/Data In 11
//     SerialComm Inputs/GVL_SDS.PCMB.stSerial1.stComIn/D @bit 96 <-> COM TxPDO-Map Inputs Channel 1/Data In 12
//     SerialComm Inputs/GVL_SDS.PCMB.stSerial1.stComIn/D @bit 104 <-> COM TxPDO-Map Inputs Channel 1/Data In 13
//     SerialComm Inputs/GVL_SDS.PCMB.stSerial1.stComIn/D @bit 112 <-> COM TxPDO-Map Inputs Channel 1/Data In 14
//     SerialComm Inputs/GVL_SDS.PCMB.stSerial1.stComIn/D @bit 120 <-> COM TxPDO-Map Inputs Channel 1/Data In 15
//     SerialComm Inputs/GVL_SDS.PCMB.stSerial1.stComIn/D @bit 128 <-> COM TxPDO-Map Inputs Channel 1/Data In 16
//     SerialComm Inputs/GVL_SDS.PCMB.stSerial1.stComIn/D @bit 136 <-> COM TxPDO-Map Inputs Channel 1/Data In 17
//     SerialComm Inputs/GVL_SDS.PCMB.stSerial1.stComIn/D @bit 144 <-> COM TxPDO-Map Inputs Channel 1/Data In 18
//     SerialComm Inputs/GVL_SDS.PCMB.stSerial1.stComIn/D @bit 152 <-> COM TxPDO-Map Inputs Channel 1/Data In 19
//     SerialComm Inputs/GVL_SDS.PCMB.stSerial1.stComIn/D @bit 16 <-> COM TxPDO-Map Inputs Channel 1/Data In 2
//     SerialComm Inputs/GVL_SDS.PCMB.stSerial1.stComIn/D @bit 160 <-> COM TxPDO-Map Inputs Channel 1/Data In 20
//     SerialComm Inputs/GVL_SDS.PCMB.stSerial1.stComIn/D @bit 168 <-> COM TxPDO-Map Inputs Channel 1/Data In 21
//     SerialComm Inputs/GVL_SDS.PCMB.stSerial1.stComIn/D @bit 24 <-> COM TxPDO-Map Inputs Channel 1/Data In 3
//     SerialComm Inputs/GVL_SDS.PCMB.stSerial1.stComIn/D @bit 32 <-> COM TxPDO-Map Inputs Channel 1/Data In 4
//     SerialComm Inputs/GVL_SDS.PCMB.stSerial1.stComIn/D @bit 40 <-> COM TxPDO-Map Inputs Channel 1/Data In 5
//     SerialComm Inputs/GVL_SDS.PCMB.stSerial1.stComIn/D @bit 48 <-> COM TxPDO-Map Inputs Channel 1/Data In 6
//     SerialComm Inputs/GVL_SDS.PCMB.stSerial1.stComIn/D @bit 56 <-> COM TxPDO-Map Inputs Channel 1/Data In 7
//     SerialComm Inputs/GVL_SDS.PCMB.stSerial1.stComIn/D @bit 64 <-> COM TxPDO-Map Inputs Channel 1/Data In 8
//     SerialComm Inputs/GVL_SDS.PCMB.stSerial1.stComIn/D @bit 72 <-> COM TxPDO-Map Inputs Channel 1/Data In 9
//     SerialComm Inputs/GVL_SDS.PCMB.stSerial2.stComIn/D @bit 8 <-> COM TxPDO-Map Inputs Channel 2/Data In 1
//     SerialComm Inputs/GVL_SDS.PCMB.stSerial2.stComIn/D @bit 80 <-> COM TxPDO-Map Inputs Channel 2/Data In 10
//     SerialComm Inputs/GVL_SDS.PCMB.stSerial2.stComIn/D @bit 88 <-> COM TxPDO-Map Inputs Channel 2/Data In 11
//     SerialComm Inputs/GVL_SDS.PCMB.stSerial2.stComIn/D @bit 96 <-> COM TxPDO-Map Inputs Channel 2/Data In 12
//     SerialComm Inputs/GVL_SDS.PCMB.stSerial2.stComIn/D @bit 104 <-> COM TxPDO-Map Inputs Channel 2/Data In 13
//     SerialComm Inputs/GVL_SDS.PCMB.stSerial2.stComIn/D @bit 112 <-> COM TxPDO-Map Inputs Channel 2/Data In 14
//     SerialComm Inputs/GVL_SDS.PCMB.stSerial2.stComIn/D @bit 120 <-> COM TxPDO-Map Inputs Channel 2/Data In 15
//     SerialComm Inputs/GVL_SDS.PCMB.stSerial2.stComIn/D @bit 128 <-> COM TxPDO-Map Inputs Channel 2/Data In 16
//     SerialComm Inputs/GVL_SDS.PCMB.stSerial2.stComIn/D @bit 136 <-> COM TxPDO-Map Inputs Channel 2/Data In 17
//     SerialComm Inputs/GVL_SDS.PCMB.stSerial2.stComIn/D @bit 144 <-> COM TxPDO-Map Inputs Channel 2/Data In 18
//     SerialComm Inputs/GVL_SDS.PCMB.stSerial2.stComIn/D @bit 152 <-> COM TxPDO-Map Inputs Channel 2/Data In 19
//     SerialComm Inputs/GVL_SDS.PCMB.stSerial2.stComIn/D @bit 16 <-> COM TxPDO-Map Inputs Channel 2/Data In 2
//     SerialComm Inputs/GVL_SDS.PCMB.stSerial2.stComIn/D @bit 160 <-> COM TxPDO-Map Inputs Channel 2/Data In 20
//     SerialComm Inputs/GVL_SDS.PCMB.stSerial2.stComIn/D @bit 168 <-> COM TxPDO-Map Inputs Channel 2/Data In 21
//     SerialComm Inputs/GVL_SDS.PCMB.stSerial2.stComIn/D @bit 24 <-> COM TxPDO-Map Inputs Channel 2/Data In 3
//     SerialComm Inputs/GVL_SDS.PCMB.stSerial2.stComIn/D @bit 32 <-> COM TxPDO-Map Inputs Channel 2/Data In 4
//     SerialComm Inputs/GVL_SDS.PCMB.stSerial2.stComIn/D @bit 40 <-> COM TxPDO-Map Inputs Channel 2/Data In 5
//     SerialComm Inputs/GVL_SDS.PCMB.stSerial2.stComIn/D @bit 48 <-> COM TxPDO-Map Inputs Channel 2/Data In 6
//     SerialComm Inputs/GVL_SDS.PCMB.stSerial2.stComIn/D @bit 56 <-> COM TxPDO-Map Inputs Channel 2/Data In 7
//     SerialComm Inputs/GVL_SDS.PCMB.stSerial2.stComIn/D @bit 64 <-> COM TxPDO-Map Inputs Channel 2/Data In 8
//     SerialComm Inputs/GVL_SDS.PCMB.stSerial2.stComIn/D @bit 72 <-> COM TxPDO-Map Inputs Channel 2/Data In 9
//     SerialComm Inputs/GVL_SDS.PCMB.stSerial1.stComIn/Status <-> COM TxPDO-Map Inputs Channel 1/Status
//     SerialComm Inputs/GVL_SDS.PCMB.stSerial2.stComIn/Status <-> COM TxPDO-Map Inputs Channel 2/Status
//     SerialComm Outputs/GVL_SDS.PCMB.stSerial1.stComOut/Ctrl <-> COM RxPDO-Map Outputs Channel 1/Ctrl
//     SerialComm Outputs/GVL_SDS.PCMB.stSerial2.stComOut/Ctrl <-> COM RxPDO-Map Outputs Channel 2/Ctrl
//     SerialComm Outputs/GVL_SDS.PCMB.stSerial1.stComOut/D <-> COM RxPDO-Map Outputs Channel 1/Data Out 0
//     SerialComm Outputs/GVL_SDS.PCMB.stSerial2.stComOut/D <-> COM RxPDO-Map Outputs Channel 2/Data Out 0
//     SerialComm Outputs/GVL_SDS.PCMB.stSerial1.stComOut/D @bit 8 <-> COM RxPDO-Map Outputs Channel 1/Data Out 1
//     SerialComm Outputs/GVL_SDS.PCMB.stSerial1.stComOut/D @bit 80 <-> COM RxPDO-Map Outputs Channel 1/Data Out 10
//     SerialComm Outputs/GVL_SDS.PCMB.stSerial1.stComOut/D @bit 88 <-> COM RxPDO-Map Outputs Channel 1/Data Out 11
//     SerialComm Outputs/GVL_SDS.PCMB.stSerial1.stComOut/D @bit 96 <-> COM RxPDO-Map Outputs Channel 1/Data Out 12
//     SerialComm Outputs/GVL_SDS.PCMB.stSerial1.stComOut/D @bit 104 <-> COM RxPDO-Map Outputs Channel 1/Data Out 13
//     SerialComm Outputs/GVL_SDS.PCMB.stSerial1.stComOut/D @bit 112 <-> COM RxPDO-Map Outputs Channel 1/Data Out 14
//     SerialComm Outputs/GVL_SDS.PCMB.stSerial1.stComOut/D @bit 120 <-> COM RxPDO-Map Outputs Channel 1/Data Out 15
//     SerialComm Outputs/GVL_SDS.PCMB.stSerial1.stComOut/D @bit 128 <-> COM RxPDO-Map Outputs Channel 1/Data Out 16
//     SerialComm Outputs/GVL_SDS.PCMB.stSerial1.stComOut/D @bit 136 <-> COM RxPDO-Map Outputs Channel 1/Data Out 17
//     SerialComm Outputs/GVL_SDS.PCMB.stSerial1.stComOut/D @bit 144 <-> COM RxPDO-Map Outputs Channel 1/Data Out 18
//     SerialComm Outputs/GVL_SDS.PCMB.stSerial1.stComOut/D @bit 152 <-> COM RxPDO-Map Outputs Channel 1/Data Out 19
//     SerialComm Outputs/GVL_SDS.PCMB.stSerial1.stComOut/D @bit 16 <-> COM RxPDO-Map Outputs Channel 1/Data Out 2
//     SerialComm Outputs/GVL_SDS.PCMB.stSerial1.stComOut/D @bit 160 <-> COM RxPDO-Map Outputs Channel 1/Data Out 20
//     SerialComm Outputs/GVL_SDS.PCMB.stSerial1.stComOut/D @bit 168 <-> COM RxPDO-Map Outputs Channel 1/Data Out 21
//     SerialComm Outputs/GVL_SDS.PCMB.stSerial1.stComOut/D @bit 24 <-> COM RxPDO-Map Outputs Channel 1/Data Out 3
//     SerialComm Outputs/GVL_SDS.PCMB.stSerial1.stComOut/D @bit 32 <-> COM RxPDO-Map Outputs Channel 1/Data Out 4
//     SerialComm Outputs/GVL_SDS.PCMB.stSerial1.stComOut/D @bit 40 <-> COM RxPDO-Map Outputs Channel 1/Data Out 5
//     SerialComm Outputs/GVL_SDS.PCMB.stSerial1.stComOut/D @bit 48 <-> COM RxPDO-Map Outputs Channel 1/Data Out 6
//     SerialComm Outputs/GVL_SDS.PCMB.stSerial1.stComOut/D @bit 56 <-> COM RxPDO-Map Outputs Channel 1/Data Out 7
//     SerialComm Outputs/GVL_SDS.PCMB.stSerial1.stComOut/D @bit 64 <-> COM RxPDO-Map Outputs Channel 1/Data Out 8
//     SerialComm Outputs/GVL_SDS.PCMB.stSerial1.stComOut/D @bit 72 <-> COM RxPDO-Map Outputs Channel 1/Data Out 9
//     SerialComm Outputs/GVL_SDS.PCMB.stSerial2.stComOut/D @bit 8 <-> COM RxPDO-Map Outputs Channel 2/Data Out 1
//     SerialComm Outputs/GVL_SDS.PCMB.stSerial2.stComOut/D @bit 80 <-> COM RxPDO-Map Outputs Channel 2/Data Out 10
//     SerialComm Outputs/GVL_SDS.PCMB.stSerial2.stComOut/D @bit 88 <-> COM RxPDO-Map Outputs Channel 2/Data Out 11
//     SerialComm Outputs/GVL_SDS.PCMB.stSerial2.stComOut/D @bit 96 <-> COM RxPDO-Map Outputs Channel 2/Data Out 12
//     SerialComm Outputs/GVL_SDS.PCMB.stSerial2.stComOut/D @bit 104 <-> COM RxPDO-Map Outputs Channel 2/Data Out 13
//     SerialComm Outputs/GVL_SDS.PCMB.stSerial2.stComOut/D @bit 112 <-> COM RxPDO-Map Outputs Channel 2/Data Out 14
//     SerialComm Outputs/GVL_SDS.PCMB.stSerial2.stComOut/D @bit 120 <-> COM RxPDO-Map Outputs Channel 2/Data Out 15
//     SerialComm Outputs/GVL_SDS.PCMB.stSerial2.stComOut/D @bit 128 <-> COM RxPDO-Map Outputs Channel 2/Data Out 16
//     SerialComm Outputs/GVL_SDS.PCMB.stSerial2.stComOut/D @bit 136 <-> COM RxPDO-Map Outputs Channel 2/Data Out 17
//     SerialComm Outputs/GVL_SDS.PCMB.stSerial2.stComOut/D @bit 144 <-> COM RxPDO-Map Outputs Channel 2/Data Out 18
//     SerialComm Outputs/GVL_SDS.PCMB.stSerial2.stComOut/D @bit 152 <-> COM RxPDO-Map Outputs Channel 2/Data Out 19
//     SerialComm Outputs/GVL_SDS.PCMB.stSerial2.stComOut/D @bit 16 <-> COM RxPDO-Map Outputs Channel 2/Data Out 2
//     SerialComm Outputs/GVL_SDS.PCMB.stSerial2.stComOut/D @bit 160 <-> COM RxPDO-Map Outputs Channel 2/Data Out 20
//     SerialComm Outputs/GVL_SDS.PCMB.stSerial2.stComOut/D @bit 168 <-> COM RxPDO-Map Outputs Channel 2/Data Out 21
//     SerialComm Outputs/GVL_SDS.PCMB.stSerial2.stComOut/D @bit 24 <-> COM RxPDO-Map Outputs Channel 2/Data Out 3
//     SerialComm Outputs/GVL_SDS.PCMB.stSerial2.stComOut/D @bit 32 <-> COM RxPDO-Map Outputs Channel 2/Data Out 4
//     SerialComm Outputs/GVL_SDS.PCMB.stSerial2.stComOut/D @bit 40 <-> COM RxPDO-Map Outputs Channel 2/Data Out 5
//     SerialComm Outputs/GVL_SDS.PCMB.stSerial2.stComOut/D @bit 48 <-> COM RxPDO-Map Outputs Channel 2/Data Out 6
//     SerialComm Outputs/GVL_SDS.PCMB.stSerial2.stComOut/D @bit 56 <-> COM RxPDO-Map Outputs Channel 2/Data Out 7
//     SerialComm Outputs/GVL_SDS.PCMB.stSerial2.stComOut/D @bit 64 <-> COM RxPDO-Map Outputs Channel 2/Data Out 8
//     SerialComm Outputs/GVL_SDS.PCMB.stSerial2.stComOut/D @bit 72 <-> COM RxPDO-Map Outputs Channel 2/Data Out 9
//   sample_delivery Instance <-> MAIN (EtherCAT)/PCM C (EP1111)
//     PlcTask Inputs/GVL_SDS.PCMC.stBaseIO.i_SyncUnitWC <-> WcState/WcState
//   sample_delivery Instance <-> MAIN (EtherCAT)/PCM C (EP4374-0002)
//     PlcTask Inputs/GVL_SDS.PCMC.stPropAir1.i_iPressRB <-> AI Inputs Channel 1/Value
//     PlcTask Inputs/GVL_SDS.PCMC.stPropAir2.i_iPressRB <-> AI Inputs Channel 2/Value
//     PlcTask Outputs/GVL_SDS.PCMC.stPropAir1.q_iPressCt <-> AO Outputs Channel 3/Analog output
//     PlcTask Outputs/GVL_SDS.PCMC.stPropAir2.q_iPressCt <-> AO Outputs Channel 4/Analog output
//   sample_delivery Instance <-> MAIN (EtherCAT)/PCM C (EP6002-0002)
//     SerialComm Inputs/GVL_SDS.PCMC.stSerial1.stComIn/D <-> COM TxPDO-Map Inputs Channel 1/Data In 0
//     SerialComm Inputs/GVL_SDS.PCMC.stSerial2.stComIn/D <-> COM TxPDO-Map Inputs Channel 2/Data In 0
//     SerialComm Inputs/GVL_SDS.PCMC.stSerial1.stComIn/D @bit 8 <-> COM TxPDO-Map Inputs Channel 1/Data In 1
//     SerialComm Inputs/GVL_SDS.PCMC.stSerial1.stComIn/D @bit 80 <-> COM TxPDO-Map Inputs Channel 1/Data In 10
//     SerialComm Inputs/GVL_SDS.PCMC.stSerial1.stComIn/D @bit 88 <-> COM TxPDO-Map Inputs Channel 1/Data In 11
//     SerialComm Inputs/GVL_SDS.PCMC.stSerial1.stComIn/D @bit 96 <-> COM TxPDO-Map Inputs Channel 1/Data In 12
//     SerialComm Inputs/GVL_SDS.PCMC.stSerial1.stComIn/D @bit 104 <-> COM TxPDO-Map Inputs Channel 1/Data In 13
//     SerialComm Inputs/GVL_SDS.PCMC.stSerial1.stComIn/D @bit 112 <-> COM TxPDO-Map Inputs Channel 1/Data In 14
//     SerialComm Inputs/GVL_SDS.PCMC.stSerial1.stComIn/D @bit 120 <-> COM TxPDO-Map Inputs Channel 1/Data In 15
//     SerialComm Inputs/GVL_SDS.PCMC.stSerial1.stComIn/D @bit 128 <-> COM TxPDO-Map Inputs Channel 1/Data In 16
//     SerialComm Inputs/GVL_SDS.PCMC.stSerial1.stComIn/D @bit 136 <-> COM TxPDO-Map Inputs Channel 1/Data In 17
//     SerialComm Inputs/GVL_SDS.PCMC.stSerial1.stComIn/D @bit 144 <-> COM TxPDO-Map Inputs Channel 1/Data In 18
//     SerialComm Inputs/GVL_SDS.PCMC.stSerial1.stComIn/D @bit 152 <-> COM TxPDO-Map Inputs Channel 1/Data In 19
//     SerialComm Inputs/GVL_SDS.PCMC.stSerial1.stComIn/D @bit 16 <-> COM TxPDO-Map Inputs Channel 1/Data In 2
//     SerialComm Inputs/GVL_SDS.PCMC.stSerial1.stComIn/D @bit 160 <-> COM TxPDO-Map Inputs Channel 1/Data In 20
//     SerialComm Inputs/GVL_SDS.PCMC.stSerial1.stComIn/D @bit 168 <-> COM TxPDO-Map Inputs Channel 1/Data In 21
//     SerialComm Inputs/GVL_SDS.PCMC.stSerial1.stComIn/D @bit 24 <-> COM TxPDO-Map Inputs Channel 1/Data In 3
//     SerialComm Inputs/GVL_SDS.PCMC.stSerial1.stComIn/D @bit 32 <-> COM TxPDO-Map Inputs Channel 1/Data In 4
//     SerialComm Inputs/GVL_SDS.PCMC.stSerial1.stComIn/D @bit 40 <-> COM TxPDO-Map Inputs Channel 1/Data In 5
//     SerialComm Inputs/GVL_SDS.PCMC.stSerial1.stComIn/D @bit 48 <-> COM TxPDO-Map Inputs Channel 1/Data In 6
//     SerialComm Inputs/GVL_SDS.PCMC.stSerial1.stComIn/D @bit 56 <-> COM TxPDO-Map Inputs Channel 1/Data In 7
//     SerialComm Inputs/GVL_SDS.PCMC.stSerial1.stComIn/D @bit 64 <-> COM TxPDO-Map Inputs Channel 1/Data In 8
//     SerialComm Inputs/GVL_SDS.PCMC.stSerial1.stComIn/D @bit 72 <-> COM TxPDO-Map Inputs Channel 1/Data In 9
//     SerialComm Inputs/GVL_SDS.PCMC.stSerial2.stComIn/D @bit 8 <-> COM TxPDO-Map Inputs Channel 2/Data In 1
//     SerialComm Inputs/GVL_SDS.PCMC.stSerial2.stComIn/D @bit 80 <-> COM TxPDO-Map Inputs Channel 2/Data In 10
//     SerialComm Inputs/GVL_SDS.PCMC.stSerial2.stComIn/D @bit 88 <-> COM TxPDO-Map Inputs Channel 2/Data In 11
//     SerialComm Inputs/GVL_SDS.PCMC.stSerial2.stComIn/D @bit 96 <-> COM TxPDO-Map Inputs Channel 2/Data In 12
//     SerialComm Inputs/GVL_SDS.PCMC.stSerial2.stComIn/D @bit 104 <-> COM TxPDO-Map Inputs Channel 2/Data In 13
//     SerialComm Inputs/GVL_SDS.PCMC.stSerial2.stComIn/D @bit 112 <-> COM TxPDO-Map Inputs Channel 2/Data In 14
//     SerialComm Inputs/GVL_SDS.PCMC.stSerial2.stComIn/D @bit 120 <-> COM TxPDO-Map Inputs Channel 2/Data In 15
//     SerialComm Inputs/GVL_SDS.PCMC.stSerial2.stComIn/D @bit 128 <-> COM TxPDO-Map Inputs Channel 2/Data In 16
//     SerialComm Inputs/GVL_SDS.PCMC.stSerial2.stComIn/D @bit 136 <-> COM TxPDO-Map Inputs Channel 2/Data In 17
//     SerialComm Inputs/GVL_SDS.PCMC.stSerial2.stComIn/D @bit 144 <-> COM TxPDO-Map Inputs Channel 2/Data In 18
//     SerialComm Inputs/GVL_SDS.PCMC.stSerial2.stComIn/D @bit 152 <-> COM TxPDO-Map Inputs Channel 2/Data In 19
//     SerialComm Inputs/GVL_SDS.PCMC.stSerial2.stComIn/D @bit 16 <-> COM TxPDO-Map Inputs Channel 2/Data In 2
//     SerialComm Inputs/GVL_SDS.PCMC.stSerial2.stComIn/D @bit 160 <-> COM TxPDO-Map Inputs Channel 2/Data In 20
//     SerialComm Inputs/GVL_SDS.PCMC.stSerial2.stComIn/D @bit 168 <-> COM TxPDO-Map Inputs Channel 2/Data In 21
//     SerialComm Inputs/GVL_SDS.PCMC.stSerial2.stComIn/D @bit 24 <-> COM TxPDO-Map Inputs Channel 2/Data In 3
//     SerialComm Inputs/GVL_SDS.PCMC.stSerial2.stComIn/D @bit 32 <-> COM TxPDO-Map Inputs Channel 2/Data In 4
//     SerialComm Inputs/GVL_SDS.PCMC.stSerial2.stComIn/D @bit 40 <-> COM TxPDO-Map Inputs Channel 2/Data In 5
//     SerialComm Inputs/GVL_SDS.PCMC.stSerial2.stComIn/D @bit 48 <-> COM TxPDO-Map Inputs Channel 2/Data In 6
//     SerialComm Inputs/GVL_SDS.PCMC.stSerial2.stComIn/D @bit 56 <-> COM TxPDO-Map Inputs Channel 2/Data In 7
//     SerialComm Inputs/GVL_SDS.PCMC.stSerial2.stComIn/D @bit 64 <-> COM TxPDO-Map Inputs Channel 2/Data In 8
//     SerialComm Inputs/GVL_SDS.PCMC.stSerial2.stComIn/D @bit 72 <-> COM TxPDO-Map Inputs Channel 2/Data In 9
//     SerialComm Inputs/GVL_SDS.PCMC.stSerial1.stComIn/Status <-> COM TxPDO-Map Inputs Channel 1/Status
//     SerialComm Inputs/GVL_SDS.PCMC.stSerial2.stComIn/Status <-> COM TxPDO-Map Inputs Channel 2/Status
//     SerialComm Outputs/GVL_SDS.PCMC.stSerial1.stComOut/Ctrl <-> COM RxPDO-Map Outputs Channel 1/Ctrl
//     SerialComm Outputs/GVL_SDS.PCMC.stSerial2.stComOut/Ctrl <-> COM RxPDO-Map Outputs Channel 2/Ctrl
//     SerialComm Outputs/GVL_SDS.PCMC.stSerial1.stComOut/D <-> COM RxPDO-Map Outputs Channel 1/Data Out 0
//     SerialComm Outputs/GVL_SDS.PCMC.stSerial2.stComOut/D <-> COM RxPDO-Map Outputs Channel 2/Data Out 0
//     SerialComm Outputs/GVL_SDS.PCMC.stSerial1.stComOut/D @bit 8 <-> COM RxPDO-Map Outputs Channel 1/Data Out 1
//     SerialComm Outputs/GVL_SDS.PCMC.stSerial1.stComOut/D @bit 80 <-> COM RxPDO-Map Outputs Channel 1/Data Out 10
//     SerialComm Outputs/GVL_SDS.PCMC.stSerial1.stComOut/D @bit 88 <-> COM RxPDO-Map Outputs Channel 1/Data Out 11
//     SerialComm Outputs/GVL_SDS.PCMC.stSerial1.stComOut/D @bit 96 <-> COM RxPDO-Map Outputs Channel 1/Data Out 12
//     SerialComm Outputs/GVL_SDS.PCMC.stSerial1.stComOut/D @bit 104 <-> COM RxPDO-Map Outputs Channel 1/Data Out 13
//     SerialComm Outputs/GVL_SDS.PCMC.stSerial1.stComOut/D @bit 112 <-> COM RxPDO-Map Outputs Channel 1/Data Out 14
//     SerialComm Outputs/GVL_SDS.PCMC.stSerial1.stComOut/D @bit 120 <-> COM RxPDO-Map Outputs Channel 1/Data Out 15
//     SerialComm Outputs/GVL_SDS.PCMC.stSerial1.stComOut/D @bit 128 <-> COM RxPDO-Map Outputs Channel 1/Data Out 16
//     SerialComm Outputs/GVL_SDS.PCMC.stSerial1.stComOut/D @bit 136 <-> COM RxPDO-Map Outputs Channel 1/Data Out 17
//     SerialComm Outputs/GVL_SDS.PCMC.stSerial1.stComOut/D @bit 144 <-> COM RxPDO-Map Outputs Channel 1/Data Out 18
//     SerialComm Outputs/GVL_SDS.PCMC.stSerial1.stComOut/D @bit 152 <-> COM RxPDO-Map Outputs Channel 1/Data Out 19
//     SerialComm Outputs/GVL_SDS.PCMC.stSerial1.stComOut/D @bit 16 <-> COM RxPDO-Map Outputs Channel 1/Data Out 2
//     SerialComm Outputs/GVL_SDS.PCMC.stSerial1.stComOut/D @bit 160 <-> COM RxPDO-Map Outputs Channel 1/Data Out 20
//     SerialComm Outputs/GVL_SDS.PCMC.stSerial1.stComOut/D @bit 168 <-> COM RxPDO-Map Outputs Channel 1/Data Out 21
//     SerialComm Outputs/GVL_SDS.PCMC.stSerial1.stComOut/D @bit 24 <-> COM RxPDO-Map Outputs Channel 1/Data Out 3
//     SerialComm Outputs/GVL_SDS.PCMC.stSerial1.stComOut/D @bit 32 <-> COM RxPDO-Map Outputs Channel 1/Data Out 4
//     SerialComm Outputs/GVL_SDS.PCMC.stSerial1.stComOut/D @bit 40 <-> COM RxPDO-Map Outputs Channel 1/Data Out 5
//     SerialComm Outputs/GVL_SDS.PCMC.stSerial1.stComOut/D @bit 48 <-> COM RxPDO-Map Outputs Channel 1/Data Out 6
//     SerialComm Outputs/GVL_SDS.PCMC.stSerial1.stComOut/D @bit 56 <-> COM RxPDO-Map Outputs Channel 1/Data Out 7
//     SerialComm Outputs/GVL_SDS.PCMC.stSerial1.stComOut/D @bit 64 <-> COM RxPDO-Map Outputs Channel 1/Data Out 8
//     SerialComm Outputs/GVL_SDS.PCMC.stSerial1.stComOut/D @bit 72 <-> COM RxPDO-Map Outputs Channel 1/Data Out 9
//     SerialComm Outputs/GVL_SDS.PCMC.stSerial2.stComOut/D @bit 8 <-> COM RxPDO-Map Outputs Channel 2/Data Out 1
//     SerialComm Outputs/GVL_SDS.PCMC.stSerial2.stComOut/D @bit 80 <-> COM RxPDO-Map Outputs Channel 2/Data Out 10
//     SerialComm Outputs/GVL_SDS.PCMC.stSerial2.stComOut/D @bit 88 <-> COM RxPDO-Map Outputs Channel 2/Data Out 11
//     SerialComm Outputs/GVL_SDS.PCMC.stSerial2.stComOut/D @bit 96 <-> COM RxPDO-Map Outputs Channel 2/Data Out 12
//     SerialComm Outputs/GVL_SDS.PCMC.stSerial2.stComOut/D @bit 104 <-> COM RxPDO-Map Outputs Channel 2/Data Out 13
//     SerialComm Outputs/GVL_SDS.PCMC.stSerial2.stComOut/D @bit 112 <-> COM RxPDO-Map Outputs Channel 2/Data Out 14
//     SerialComm Outputs/GVL_SDS.PCMC.stSerial2.stComOut/D @bit 120 <-> COM RxPDO-Map Outputs Channel 2/Data Out 15
//     SerialComm Outputs/GVL_SDS.PCMC.stSerial2.stComOut/D @bit 128 <-> COM RxPDO-Map Outputs Channel 2/Data Out 16
//     SerialComm Outputs/GVL_SDS.PCMC.stSerial2.stComOut/D @bit 136 <-> COM RxPDO-Map Outputs Channel 2/Data Out 17
//     SerialComm Outputs/GVL_SDS.PCMC.stSerial2.stComOut/D @bit 144 <-> COM RxPDO-Map Outputs Channel 2/Data Out 18
//     SerialComm Outputs/GVL_SDS.PCMC.stSerial2.stComOut/D @bit 152 <-> COM RxPDO-Map Outputs Channel 2/Data Out 19
//     SerialComm Outputs/GVL_SDS.PCMC.stSerial2.stComOut/D @bit 16 <-> COM RxPDO-Map Outputs Channel 2/Data Out 2
//     SerialComm Outputs/GVL_SDS.PCMC.stSerial2.stComOut/D @bit 160 <-> COM RxPDO-Map Outputs Channel 2/Data Out 20
//     SerialComm Outputs/GVL_SDS.PCMC.stSerial2.stComOut/D @bit 168 <-> COM RxPDO-Map Outputs Channel 2/Data Out 21
//     SerialComm Outputs/GVL_SDS.PCMC.stSerial2.stComOut/D @bit 24 <-> COM RxPDO-Map Outputs Channel 2/Data Out 3
//     SerialComm Outputs/GVL_SDS.PCMC.stSerial2.stComOut/D @bit 32 <-> COM RxPDO-Map Outputs Channel 2/Data Out 4
//     SerialComm Outputs/GVL_SDS.PCMC.stSerial2.stComOut/D @bit 40 <-> COM RxPDO-Map Outputs Channel 2/Data Out 5
//     SerialComm Outputs/GVL_SDS.PCMC.stSerial2.stComOut/D @bit 48 <-> COM RxPDO-Map Outputs Channel 2/Data Out 6
//     SerialComm Outputs/GVL_SDS.PCMC.stSerial2.stComOut/D @bit 56 <-> COM RxPDO-Map Outputs Channel 2/Data Out 7
//     SerialComm Outputs/GVL_SDS.PCMC.stSerial2.stComOut/D @bit 64 <-> COM RxPDO-Map Outputs Channel 2/Data Out 8
//     SerialComm Outputs/GVL_SDS.PCMC.stSerial2.stComOut/D @bit 72 <-> COM RxPDO-Map Outputs Channel 2/Data Out 9
//   sample_delivery Instance <-> MAIN (EtherCAT)/PCM D (EP1111)
//     PlcTask Inputs/GVL_SDS.PCMD.stBaseIO.i_SyncUnitWC <-> WcState/WcState
//   sample_delivery Instance <-> MAIN (EtherCAT)/PCM D (EP4374-0002)
//     PlcTask Inputs/GVL_SDS.PCMD.stPropAir1.i_iPressRB <-> AI Inputs Channel 1/Value
//     PlcTask Inputs/GVL_SDS.PCMD.stPropAir2.i_iPressRB <-> AI Inputs Channel 2/Value
//     PlcTask Outputs/GVL_SDS.PCMD.stPropAir1.q_iPressCt <-> AO Outputs Channel 3/Analog output
//     PlcTask Outputs/GVL_SDS.PCMD.stPropAir2.q_iPressCt <-> AO Outputs Channel 4/Analog output
//   sample_delivery Instance <-> MAIN (EtherCAT)/PCM D (EP6002-0002)
//     SerialComm Inputs/GVL_SDS.PCMD.stSerial1.stComIn/D <-> COM TxPDO-Map Inputs Channel 1/Data In 0
//     SerialComm Inputs/GVL_SDS.PCMD.stSerial2.stComIn/D <-> COM TxPDO-Map Inputs Channel 2/Data In 0
//     SerialComm Inputs/GVL_SDS.PCMD.stSerial1.stComIn/D @bit 8 <-> COM TxPDO-Map Inputs Channel 1/Data In 1
//     SerialComm Inputs/GVL_SDS.PCMD.stSerial1.stComIn/D @bit 80 <-> COM TxPDO-Map Inputs Channel 1/Data In 10
//     SerialComm Inputs/GVL_SDS.PCMD.stSerial1.stComIn/D @bit 88 <-> COM TxPDO-Map Inputs Channel 1/Data In 11
//     SerialComm Inputs/GVL_SDS.PCMD.stSerial1.stComIn/D @bit 96 <-> COM TxPDO-Map Inputs Channel 1/Data In 12
//     SerialComm Inputs/GVL_SDS.PCMD.stSerial1.stComIn/D @bit 104 <-> COM TxPDO-Map Inputs Channel 1/Data In 13
//     SerialComm Inputs/GVL_SDS.PCMD.stSerial1.stComIn/D @bit 112 <-> COM TxPDO-Map Inputs Channel 1/Data In 14
//     SerialComm Inputs/GVL_SDS.PCMD.stSerial1.stComIn/D @bit 120 <-> COM TxPDO-Map Inputs Channel 1/Data In 15
//     SerialComm Inputs/GVL_SDS.PCMD.stSerial1.stComIn/D @bit 128 <-> COM TxPDO-Map Inputs Channel 1/Data In 16
//     SerialComm Inputs/GVL_SDS.PCMD.stSerial1.stComIn/D @bit 136 <-> COM TxPDO-Map Inputs Channel 1/Data In 17
//     SerialComm Inputs/GVL_SDS.PCMD.stSerial1.stComIn/D @bit 144 <-> COM TxPDO-Map Inputs Channel 1/Data In 18
//     SerialComm Inputs/GVL_SDS.PCMD.stSerial1.stComIn/D @bit 152 <-> COM TxPDO-Map Inputs Channel 1/Data In 19
//     SerialComm Inputs/GVL_SDS.PCMD.stSerial1.stComIn/D @bit 16 <-> COM TxPDO-Map Inputs Channel 1/Data In 2
//     SerialComm Inputs/GVL_SDS.PCMD.stSerial1.stComIn/D @bit 160 <-> COM TxPDO-Map Inputs Channel 1/Data In 20
//     SerialComm Inputs/GVL_SDS.PCMD.stSerial1.stComIn/D @bit 168 <-> COM TxPDO-Map Inputs Channel 1/Data In 21
//     SerialComm Inputs/GVL_SDS.PCMD.stSerial1.stComIn/D @bit 24 <-> COM TxPDO-Map Inputs Channel 1/Data In 3
//     SerialComm Inputs/GVL_SDS.PCMD.stSerial1.stComIn/D @bit 32 <-> COM TxPDO-Map Inputs Channel 1/Data In 4
//     SerialComm Inputs/GVL_SDS.PCMD.stSerial1.stComIn/D @bit 40 <-> COM TxPDO-Map Inputs Channel 1/Data In 5
//     SerialComm Inputs/GVL_SDS.PCMD.stSerial1.stComIn/D @bit 48 <-> COM TxPDO-Map Inputs Channel 1/Data In 6
//     SerialComm Inputs/GVL_SDS.PCMD.stSerial1.stComIn/D @bit 56 <-> COM TxPDO-Map Inputs Channel 1/Data In 7
//     SerialComm Inputs/GVL_SDS.PCMD.stSerial1.stComIn/D @bit 64 <-> COM TxPDO-Map Inputs Channel 1/Data In 8
//     SerialComm Inputs/GVL_SDS.PCMD.stSerial1.stComIn/D @bit 72 <-> COM TxPDO-Map Inputs Channel 1/Data In 9
//     SerialComm Inputs/GVL_SDS.PCMD.stSerial2.stComIn/D @bit 8 <-> COM TxPDO-Map Inputs Channel 2/Data In 1
//     SerialComm Inputs/GVL_SDS.PCMD.stSerial2.stComIn/D @bit 80 <-> COM TxPDO-Map Inputs Channel 2/Data In 10
//     SerialComm Inputs/GVL_SDS.PCMD.stSerial2.stComIn/D @bit 88 <-> COM TxPDO-Map Inputs Channel 2/Data In 11
//     SerialComm Inputs/GVL_SDS.PCMD.stSerial2.stComIn/D @bit 96 <-> COM TxPDO-Map Inputs Channel 2/Data In 12
//     SerialComm Inputs/GVL_SDS.PCMD.stSerial2.stComIn/D @bit 104 <-> COM TxPDO-Map Inputs Channel 2/Data In 13
//     SerialComm Inputs/GVL_SDS.PCMD.stSerial2.stComIn/D @bit 112 <-> COM TxPDO-Map Inputs Channel 2/Data In 14
//     SerialComm Inputs/GVL_SDS.PCMD.stSerial2.stComIn/D @bit 120 <-> COM TxPDO-Map Inputs Channel 2/Data In 15
//     SerialComm Inputs/GVL_SDS.PCMD.stSerial2.stComIn/D @bit 128 <-> COM TxPDO-Map Inputs Channel 2/Data In 16
//     SerialComm Inputs/GVL_SDS.PCMD.stSerial2.stComIn/D @bit 136 <-> COM TxPDO-Map Inputs Channel 2/Data In 17
//     SerialComm Inputs/GVL_SDS.PCMD.stSerial2.stComIn/D @bit 144 <-> COM TxPDO-Map Inputs Channel 2/Data In 18
//     SerialComm Inputs/GVL_SDS.PCMD.stSerial2.stComIn/D @bit 152 <-> COM TxPDO-Map Inputs Channel 2/Data In 19
//     SerialComm Inputs/GVL_SDS.PCMD.stSerial2.stComIn/D @bit 16 <-> COM TxPDO-Map Inputs Channel 2/Data In 2
//     SerialComm Inputs/GVL_SDS.PCMD.stSerial2.stComIn/D @bit 160 <-> COM TxPDO-Map Inputs Channel 2/Data In 20
//     SerialComm Inputs/GVL_SDS.PCMD.stSerial2.stComIn/D @bit 168 <-> COM TxPDO-Map Inputs Channel 2/Data In 21
//     SerialComm Inputs/GVL_SDS.PCMD.stSerial2.stComIn/D @bit 24 <-> COM TxPDO-Map Inputs Channel 2/Data In 3
//     SerialComm Inputs/GVL_SDS.PCMD.stSerial2.stComIn/D @bit 32 <-> COM TxPDO-Map Inputs Channel 2/Data In 4
//     SerialComm Inputs/GVL_SDS.PCMD.stSerial2.stComIn/D @bit 40 <-> COM TxPDO-Map Inputs Channel 2/Data In 5
//     SerialComm Inputs/GVL_SDS.PCMD.stSerial2.stComIn/D @bit 48 <-> COM TxPDO-Map Inputs Channel 2/Data In 6
//     SerialComm Inputs/GVL_SDS.PCMD.stSerial2.stComIn/D @bit 56 <-> COM TxPDO-Map Inputs Channel 2/Data In 7
//     SerialComm Inputs/GVL_SDS.PCMD.stSerial2.stComIn/D @bit 64 <-> COM TxPDO-Map Inputs Channel 2/Data In 8
//     SerialComm Inputs/GVL_SDS.PCMD.stSerial2.stComIn/D @bit 72 <-> COM TxPDO-Map Inputs Channel 2/Data In 9
//     SerialComm Inputs/GVL_SDS.PCMD.stSerial1.stComIn/Status <-> COM TxPDO-Map Inputs Channel 1/Status
//     SerialComm Inputs/GVL_SDS.PCMD.stSerial2.stComIn/Status <-> COM TxPDO-Map Inputs Channel 2/Status
//     SerialComm Outputs/GVL_SDS.PCMD.stSerial1.stComOut/Ctrl <-> COM RxPDO-Map Outputs Channel 1/Ctrl
//     SerialComm Outputs/GVL_SDS.PCMD.stSerial2.stComOut/Ctrl <-> COM RxPDO-Map Outputs Channel 2/Ctrl
//     SerialComm Outputs/GVL_SDS.PCMD.stSerial1.stComOut/D <-> COM RxPDO-Map Outputs Channel 1/Data Out 0
//     SerialComm Outputs/GVL_SDS.PCMD.stSerial2.stComOut/D <-> COM RxPDO-Map Outputs Channel 2/Data Out 0
//     SerialComm Outputs/GVL_SDS.PCMD.stSerial1.stComOut/D @bit 8 <-> COM RxPDO-Map Outputs Channel 1/Data Out 1
//     SerialComm Outputs/GVL_SDS.PCMD.stSerial1.stComOut/D @bit 80 <-> COM RxPDO-Map Outputs Channel 1/Data Out 10
//     SerialComm Outputs/GVL_SDS.PCMD.stSerial1.stComOut/D @bit 88 <-> COM RxPDO-Map Outputs Channel 1/Data Out 11
//     SerialComm Outputs/GVL_SDS.PCMD.stSerial1.stComOut/D @bit 96 <-> COM RxPDO-Map Outputs Channel 1/Data Out 12
//     SerialComm Outputs/GVL_SDS.PCMD.stSerial1.stComOut/D @bit 104 <-> COM RxPDO-Map Outputs Channel 1/Data Out 13
//     SerialComm Outputs/GVL_SDS.PCMD.stSerial1.stComOut/D @bit 112 <-> COM RxPDO-Map Outputs Channel 1/Data Out 14
//     SerialComm Outputs/GVL_SDS.PCMD.stSerial1.stComOut/D @bit 120 <-> COM RxPDO-Map Outputs Channel 1/Data Out 15
//     SerialComm Outputs/GVL_SDS.PCMD.stSerial1.stComOut/D @bit 128 <-> COM RxPDO-Map Outputs Channel 1/Data Out 16
//     SerialComm Outputs/GVL_SDS.PCMD.stSerial1.stComOut/D @bit 136 <-> COM RxPDO-Map Outputs Channel 1/Data Out 17
//     SerialComm Outputs/GVL_SDS.PCMD.stSerial1.stComOut/D @bit 144 <-> COM RxPDO-Map Outputs Channel 1/Data Out 18
//     SerialComm Outputs/GVL_SDS.PCMD.stSerial1.stComOut/D @bit 152 <-> COM RxPDO-Map Outputs Channel 1/Data Out 19
//     SerialComm Outputs/GVL_SDS.PCMD.stSerial1.stComOut/D @bit 16 <-> COM RxPDO-Map Outputs Channel 1/Data Out 2
//     SerialComm Outputs/GVL_SDS.PCMD.stSerial1.stComOut/D @bit 160 <-> COM RxPDO-Map Outputs Channel 1/Data Out 20
//     SerialComm Outputs/GVL_SDS.PCMD.stSerial1.stComOut/D @bit 168 <-> COM RxPDO-Map Outputs Channel 1/Data Out 21
//     SerialComm Outputs/GVL_SDS.PCMD.stSerial1.stComOut/D @bit 24 <-> COM RxPDO-Map Outputs Channel 1/Data Out 3
//     SerialComm Outputs/GVL_SDS.PCMD.stSerial1.stComOut/D @bit 32 <-> COM RxPDO-Map Outputs Channel 1/Data Out 4
//     SerialComm Outputs/GVL_SDS.PCMD.stSerial1.stComOut/D @bit 40 <-> COM RxPDO-Map Outputs Channel 1/Data Out 5
//     SerialComm Outputs/GVL_SDS.PCMD.stSerial1.stComOut/D @bit 48 <-> COM RxPDO-Map Outputs Channel 1/Data Out 6
//     SerialComm Outputs/GVL_SDS.PCMD.stSerial1.stComOut/D @bit 56 <-> COM RxPDO-Map Outputs Channel 1/Data Out 7
//     SerialComm Outputs/GVL_SDS.PCMD.stSerial1.stComOut/D @bit 64 <-> COM RxPDO-Map Outputs Channel 1/Data Out 8
//     SerialComm Outputs/GVL_SDS.PCMD.stSerial1.stComOut/D @bit 72 <-> COM RxPDO-Map Outputs Channel 1/Data Out 9
//     SerialComm Outputs/GVL_SDS.PCMD.stSerial2.stComOut/D @bit 8 <-> COM RxPDO-Map Outputs Channel 2/Data Out 1
//     SerialComm Outputs/GVL_SDS.PCMD.stSerial2.stComOut/D @bit 80 <-> COM RxPDO-Map Outputs Channel 2/Data Out 10
//     SerialComm Outputs/GVL_SDS.PCMD.stSerial2.stComOut/D @bit 88 <-> COM RxPDO-Map Outputs Channel 2/Data Out 11
//     SerialComm Outputs/GVL_SDS.PCMD.stSerial2.stComOut/D @bit 96 <-> COM RxPDO-Map Outputs Channel 2/Data Out 12
//     SerialComm Outputs/GVL_SDS.PCMD.stSerial2.stComOut/D @bit 104 <-> COM RxPDO-Map Outputs Channel 2/Data Out 13
//     SerialComm Outputs/GVL_SDS.PCMD.stSerial2.stComOut/D @bit 112 <-> COM RxPDO-Map Outputs Channel 2/Data Out 14
//     SerialComm Outputs/GVL_SDS.PCMD.stSerial2.stComOut/D @bit 120 <-> COM RxPDO-Map Outputs Channel 2/Data Out 15
//     SerialComm Outputs/GVL_SDS.PCMD.stSerial2.stComOut/D @bit 128 <-> COM RxPDO-Map Outputs Channel 2/Data Out 16
//     SerialComm Outputs/GVL_SDS.PCMD.stSerial2.stComOut/D @bit 136 <-> COM RxPDO-Map Outputs Channel 2/Data Out 17
//     SerialComm Outputs/GVL_SDS.PCMD.stSerial2.stComOut/D @bit 144 <-> COM RxPDO-Map Outputs Channel 2/Data Out 18
//     SerialComm Outputs/GVL_SDS.PCMD.stSerial2.stComOut/D @bit 152 <-> COM RxPDO-Map Outputs Channel 2/Data Out 19
//     SerialComm Outputs/GVL_SDS.PCMD.stSerial2.stComOut/D @bit 16 <-> COM RxPDO-Map Outputs Channel 2/Data Out 2
//     SerialComm Outputs/GVL_SDS.PCMD.stSerial2.stComOut/D @bit 160 <-> COM RxPDO-Map Outputs Channel 2/Data Out 20
//     SerialComm Outputs/GVL_SDS.PCMD.stSerial2.stComOut/D @bit 168 <-> COM RxPDO-Map Outputs Channel 2/Data Out 21
//     SerialComm Outputs/GVL_SDS.PCMD.stSerial2.stComOut/D @bit 24 <-> COM RxPDO-Map Outputs Channel 2/Data Out 3
//     SerialComm Outputs/GVL_SDS.PCMD.stSerial2.stComOut/D @bit 32 <-> COM RxPDO-Map Outputs Channel 2/Data Out 4
//     SerialComm Outputs/GVL_SDS.PCMD.stSerial2.stComOut/D @bit 40 <-> COM RxPDO-Map Outputs Channel 2/Data Out 5
//     SerialComm Outputs/GVL_SDS.PCMD.stSerial2.stComOut/D @bit 48 <-> COM RxPDO-Map Outputs Channel 2/Data Out 6
//     SerialComm Outputs/GVL_SDS.PCMD.stSerial2.stComOut/D @bit 56 <-> COM RxPDO-Map Outputs Channel 2/Data Out 7
//     SerialComm Outputs/GVL_SDS.PCMD.stSerial2.stComOut/D @bit 64 <-> COM RxPDO-Map Outputs Channel 2/Data Out 8
//     SerialComm Outputs/GVL_SDS.PCMD.stSerial2.stComOut/D @bit 72 <-> COM RxPDO-Map Outputs Channel 2/Data Out 9
//   sample_delivery Instance <-> MAIN (EtherCAT)/Sensirion Flow Meter A Serial 01 (EP6002-0002)
//     PlcTask Inputs/GVL_SDS.fbSFM_01.stSensSerial.stComIn/D[0] <-> COM TxPDO-Map Inputs Channel 1/Data In 0
//     PlcTask Inputs/GVL_SDS.fbSFM_01.stSensSerial.stComIn/D[10] <-> COM TxPDO-Map Inputs Channel 1/Data In 10
//     PlcTask Inputs/GVL_SDS.fbSFM_01.stSensSerial.stComIn/D[11] <-> COM TxPDO-Map Inputs Channel 1/Data In 11
//     PlcTask Inputs/GVL_SDS.fbSFM_01.stSensSerial.stComIn/D[12] <-> COM TxPDO-Map Inputs Channel 1/Data In 12
//     PlcTask Inputs/GVL_SDS.fbSFM_01.stSensSerial.stComIn/D[13] <-> COM TxPDO-Map Inputs Channel 1/Data In 13
//     PlcTask Inputs/GVL_SDS.fbSFM_01.stSensSerial.stComIn/D[14] <-> COM TxPDO-Map Inputs Channel 1/Data In 14
//     PlcTask Inputs/GVL_SDS.fbSFM_01.stSensSerial.stComIn/D[15] <-> COM TxPDO-Map Inputs Channel 1/Data In 15
//     PlcTask Inputs/GVL_SDS.fbSFM_01.stSensSerial.stComIn/D[16] <-> COM TxPDO-Map Inputs Channel 1/Data In 16
//     PlcTask Inputs/GVL_SDS.fbSFM_01.stSensSerial.stComIn/D[17] <-> COM TxPDO-Map Inputs Channel 1/Data In 17
//     PlcTask Inputs/GVL_SDS.fbSFM_01.stSensSerial.stComIn/D[18] <-> COM TxPDO-Map Inputs Channel 1/Data In 18
//     PlcTask Inputs/GVL_SDS.fbSFM_01.stSensSerial.stComIn/D[19] <-> COM TxPDO-Map Inputs Channel 1/Data In 19
//     PlcTask Inputs/GVL_SDS.fbSFM_01.stSensSerial.stComIn/D[1] <-> COM TxPDO-Map Inputs Channel 1/Data In 1
//     PlcTask Inputs/GVL_SDS.fbSFM_01.stSensSerial.stComIn/D[20] <-> COM TxPDO-Map Inputs Channel 1/Data In 20
//     PlcTask Inputs/GVL_SDS.fbSFM_01.stSensSerial.stComIn/D[21] <-> COM TxPDO-Map Inputs Channel 1/Data In 21
//     PlcTask Inputs/GVL_SDS.fbSFM_01.stSensSerial.stComIn/D[2] <-> COM TxPDO-Map Inputs Channel 1/Data In 2
//     PlcTask Inputs/GVL_SDS.fbSFM_01.stSensSerial.stComIn/D[3] <-> COM TxPDO-Map Inputs Channel 1/Data In 3
//     PlcTask Inputs/GVL_SDS.fbSFM_01.stSensSerial.stComIn/D[4] <-> COM TxPDO-Map Inputs Channel 1/Data In 4
//     PlcTask Inputs/GVL_SDS.fbSFM_01.stSensSerial.stComIn/D[5] <-> COM TxPDO-Map Inputs Channel 1/Data In 5
//     PlcTask Inputs/GVL_SDS.fbSFM_01.stSensSerial.stComIn/D[6] <-> COM TxPDO-Map Inputs Channel 1/Data In 6
//     PlcTask Inputs/GVL_SDS.fbSFM_01.stSensSerial.stComIn/D[7] <-> COM TxPDO-Map Inputs Channel 1/Data In 7
//     PlcTask Inputs/GVL_SDS.fbSFM_01.stSensSerial.stComIn/D[8] <-> COM TxPDO-Map Inputs Channel 1/Data In 8
//     PlcTask Inputs/GVL_SDS.fbSFM_01.stSensSerial.stComIn/D[9] <-> COM TxPDO-Map Inputs Channel 1/Data In 9
//     PlcTask Inputs/GVL_SDS.fbSFM_01.stSensSerial.stComIn/Status <-> COM TxPDO-Map Inputs Channel 1/Status
//     PlcTask Inputs/GVL_SDS.fbSFM_02.stSensSerial.stComIn/Status <-> COM TxPDO-Map Inputs Channel 2/Status
//     PlcTask Inputs/GVL_SDS.fbSFM_02.stSensSerial.stComIn/D <-> COM TxPDO-Map Inputs Channel 2/Data In 0
//     PlcTask Inputs/GVL_SDS.fbSFM_02.stSensSerial.stComIn/D @bit 8 <-> COM TxPDO-Map Inputs Channel 2/Data In 1
//     PlcTask Inputs/GVL_SDS.fbSFM_02.stSensSerial.stComIn/D @bit 80 <-> COM TxPDO-Map Inputs Channel 2/Data In 10
//     PlcTask Inputs/GVL_SDS.fbSFM_02.stSensSerial.stComIn/D @bit 88 <-> COM TxPDO-Map Inputs Channel 2/Data In 11
//     PlcTask Inputs/GVL_SDS.fbSFM_02.stSensSerial.stComIn/D @bit 96 <-> COM TxPDO-Map Inputs Channel 2/Data In 12
//     PlcTask Inputs/GVL_SDS.fbSFM_02.stSensSerial.stComIn/D @bit 104 <-> COM TxPDO-Map Inputs Channel 2/Data In 13
//     PlcTask Inputs/GVL_SDS.fbSFM_02.stSensSerial.stComIn/D @bit 112 <-> COM TxPDO-Map Inputs Channel 2/Data In 14
//     PlcTask Inputs/GVL_SDS.fbSFM_02.stSensSerial.stComIn/D @bit 120 <-> COM TxPDO-Map Inputs Channel 2/Data In 15
//     PlcTask Inputs/GVL_SDS.fbSFM_02.stSensSerial.stComIn/D @bit 128 <-> COM TxPDO-Map Inputs Channel 2/Data In 16
//     PlcTask Inputs/GVL_SDS.fbSFM_02.stSensSerial.stComIn/D @bit 136 <-> COM TxPDO-Map Inputs Channel 2/Data In 17
//     PlcTask Inputs/GVL_SDS.fbSFM_02.stSensSerial.stComIn/D @bit 144 <-> COM TxPDO-Map Inputs Channel 2/Data In 18
//     PlcTask Inputs/GVL_SDS.fbSFM_02.stSensSerial.stComIn/D @bit 152 <-> COM TxPDO-Map Inputs Channel 2/Data In 19
//     PlcTask Inputs/GVL_SDS.fbSFM_02.stSensSerial.stComIn/D @bit 16 <-> COM TxPDO-Map Inputs Channel 2/Data In 2
//     PlcTask Inputs/GVL_SDS.fbSFM_02.stSensSerial.stComIn/D @bit 160 <-> COM TxPDO-Map Inputs Channel 2/Data In 20
//     PlcTask Inputs/GVL_SDS.fbSFM_02.stSensSerial.stComIn/D @bit 168 <-> COM TxPDO-Map Inputs Channel 2/Data In 21
//     PlcTask Inputs/GVL_SDS.fbSFM_02.stSensSerial.stComIn/D @bit 24 <-> COM TxPDO-Map Inputs Channel 2/Data In 3
//     PlcTask Inputs/GVL_SDS.fbSFM_02.stSensSerial.stComIn/D @bit 32 <-> COM TxPDO-Map Inputs Channel 2/Data In 4
//     PlcTask Inputs/GVL_SDS.fbSFM_02.stSensSerial.stComIn/D @bit 40 <-> COM TxPDO-Map Inputs Channel 2/Data In 5
//     PlcTask Inputs/GVL_SDS.fbSFM_02.stSensSerial.stComIn/D @bit 48 <-> COM TxPDO-Map Inputs Channel 2/Data In 6
//     PlcTask Inputs/GVL_SDS.fbSFM_02.stSensSerial.stComIn/D @bit 56 <-> COM TxPDO-Map Inputs Channel 2/Data In 7
//     PlcTask Inputs/GVL_SDS.fbSFM_02.stSensSerial.stComIn/D @bit 64 <-> COM TxPDO-Map Inputs Channel 2/Data In 8
//     PlcTask Inputs/GVL_SDS.fbSFM_02.stSensSerial.stComIn/D @bit 72 <-> COM TxPDO-Map Inputs Channel 2/Data In 9
//     PlcTask Outputs/GVL_SDS.fbSFM_01.stSensSerial.stComOut/Ctrl <-> COM RxPDO-Map Outputs Channel 1/Ctrl
//     PlcTask Outputs/GVL_SDS.fbSFM_02.stSensSerial.stComOut/Ctrl <-> COM RxPDO-Map Outputs Channel 2/Ctrl
//     PlcTask Outputs/GVL_SDS.fbSFM_01.stSensSerial.stComOut/D[0] <-> COM RxPDO-Map Outputs Channel 1/Data Out 0
//     PlcTask Outputs/GVL_SDS.fbSFM_01.stSensSerial.stComOut/D[10] <-> COM RxPDO-Map Outputs Channel 1/Data Out 10
//     PlcTask Outputs/GVL_SDS.fbSFM_01.stSensSerial.stComOut/D[11] <-> COM RxPDO-Map Outputs Channel 1/Data Out 11
//     PlcTask Outputs/GVL_SDS.fbSFM_01.stSensSerial.stComOut/D[12] <-> COM RxPDO-Map Outputs Channel 1/Data Out 12
//     PlcTask Outputs/GVL_SDS.fbSFM_01.stSensSerial.stComOut/D[13] <-> COM RxPDO-Map Outputs Channel 1/Data Out 13
//     PlcTask Outputs/GVL_SDS.fbSFM_01.stSensSerial.stComOut/D[14] <-> COM RxPDO-Map Outputs Channel 1/Data Out 14
//     PlcTask Outputs/GVL_SDS.fbSFM_01.stSensSerial.stComOut/D[15] <-> COM RxPDO-Map Outputs Channel 1/Data Out 15
//     PlcTask Outputs/GVL_SDS.fbSFM_01.stSensSerial.stComOut/D[16] <-> COM RxPDO-Map Outputs Channel 1/Data Out 16
//     PlcTask Outputs/GVL_SDS.fbSFM_01.stSensSerial.stComOut/D[17] <-> COM RxPDO-Map Outputs Channel 1/Data Out 17
//     PlcTask Outputs/GVL_SDS.fbSFM_01.stSensSerial.stComOut/D[18] <-> COM RxPDO-Map Outputs Channel 1/Data Out 18
//     PlcTask Outputs/GVL_SDS.fbSFM_01.stSensSerial.stComOut/D[19] <-> COM RxPDO-Map Outputs Channel 1/Data Out 19
//     PlcTask Outputs/GVL_SDS.fbSFM_01.stSensSerial.stComOut/D[1] <-> COM RxPDO-Map Outputs Channel 1/Data Out 1
//     PlcTask Outputs/GVL_SDS.fbSFM_01.stSensSerial.stComOut/D[20] <-> COM RxPDO-Map Outputs Channel 1/Data Out 20
//     PlcTask Outputs/GVL_SDS.fbSFM_01.stSensSerial.stComOut/D[21] <-> COM RxPDO-Map Outputs Channel 1/Data Out 21
//     PlcTask Outputs/GVL_SDS.fbSFM_01.stSensSerial.stComOut/D[2] <-> COM RxPDO-Map Outputs Channel 1/Data Out 2
//     PlcTask Outputs/GVL_SDS.fbSFM_01.stSensSerial.stComOut/D[3] <-> COM RxPDO-Map Outputs Channel 1/Data Out 3
//     PlcTask Outputs/GVL_SDS.fbSFM_01.stSensSerial.stComOut/D[4] <-> COM RxPDO-Map Outputs Channel 1/Data Out 4
//     PlcTask Outputs/GVL_SDS.fbSFM_01.stSensSerial.stComOut/D[5] <-> COM RxPDO-Map Outputs Channel 1/Data Out 5
//     PlcTask Outputs/GVL_SDS.fbSFM_01.stSensSerial.stComOut/D[6] <-> COM RxPDO-Map Outputs Channel 1/Data Out 6
//     PlcTask Outputs/GVL_SDS.fbSFM_01.stSensSerial.stComOut/D[7] <-> COM RxPDO-Map Outputs Channel 1/Data Out 7
//     PlcTask Outputs/GVL_SDS.fbSFM_01.stSensSerial.stComOut/D[8] <-> COM RxPDO-Map Outputs Channel 1/Data Out 8
//     PlcTask Outputs/GVL_SDS.fbSFM_01.stSensSerial.stComOut/D[9] <-> COM RxPDO-Map Outputs Channel 1/Data Out 9
//     PlcTask Outputs/GVL_SDS.fbSFM_02.stSensSerial.stComOut/D <-> COM RxPDO-Map Outputs Channel 2/Data Out 0
//     PlcTask Outputs/GVL_SDS.fbSFM_02.stSensSerial.stComOut/D @bit 8 <-> COM RxPDO-Map Outputs Channel 2/Data Out 1
//     PlcTask Outputs/GVL_SDS.fbSFM_02.stSensSerial.stComOut/D @bit 80 <-> COM RxPDO-Map Outputs Channel 2/Data Out 10
//     PlcTask Outputs/GVL_SDS.fbSFM_02.stSensSerial.stComOut/D @bit 88 <-> COM RxPDO-Map Outputs Channel 2/Data Out 11
//     PlcTask Outputs/GVL_SDS.fbSFM_02.stSensSerial.stComOut/D @bit 96 <-> COM RxPDO-Map Outputs Channel 2/Data Out 12
//     PlcTask Outputs/GVL_SDS.fbSFM_02.stSensSerial.stComOut/D @bit 104 <-> COM RxPDO-Map Outputs Channel 2/Data Out 13
//     PlcTask Outputs/GVL_SDS.fbSFM_02.stSensSerial.stComOut/D @bit 112 <-> COM RxPDO-Map Outputs Channel 2/Data Out 14
//     PlcTask Outputs/GVL_SDS.fbSFM_02.stSensSerial.stComOut/D @bit 120 <-> COM RxPDO-Map Outputs Channel 2/Data Out 15
//     PlcTask Outputs/GVL_SDS.fbSFM_02.stSensSerial.stComOut/D @bit 128 <-> COM RxPDO-Map Outputs Channel 2/Data Out 16
//     PlcTask Outputs/GVL_SDS.fbSFM_02.stSensSerial.stComOut/D @bit 136 <-> COM RxPDO-Map Outputs Channel 2/Data Out 17
//     PlcTask Outputs/GVL_SDS.fbSFM_02.stSensSerial.stComOut/D @bit 144 <-> COM RxPDO-Map Outputs Channel 2/Data Out 18
//     PlcTask Outputs/GVL_SDS.fbSFM_02.stSensSerial.stComOut/D @bit 152 <-> COM RxPDO-Map Outputs Channel 2/Data Out 19
//     PlcTask Outputs/GVL_SDS.fbSFM_02.stSensSerial.stComOut/D @bit 16 <-> COM RxPDO-Map Outputs Channel 2/Data Out 2
//     PlcTask Outputs/GVL_SDS.fbSFM_02.stSensSerial.stComOut/D @bit 160 <-> COM RxPDO-Map Outputs Channel 2/Data Out 20
//     PlcTask Outputs/GVL_SDS.fbSFM_02.stSensSerial.stComOut/D @bit 168 <-> COM RxPDO-Map Outputs Channel 2/Data Out 21
//     PlcTask Outputs/GVL_SDS.fbSFM_02.stSensSerial.stComOut/D @bit 24 <-> COM RxPDO-Map Outputs Channel 2/Data Out 3
//     PlcTask Outputs/GVL_SDS.fbSFM_02.stSensSerial.stComOut/D @bit 32 <-> COM RxPDO-Map Outputs Channel 2/Data Out 4
//     PlcTask Outputs/GVL_SDS.fbSFM_02.stSensSerial.stComOut/D @bit 40 <-> COM RxPDO-Map Outputs Channel 2/Data Out 5
//     PlcTask Outputs/GVL_SDS.fbSFM_02.stSensSerial.stComOut/D @bit 48 <-> COM RxPDO-Map Outputs Channel 2/Data Out 6
//     PlcTask Outputs/GVL_SDS.fbSFM_02.stSensSerial.stComOut/D @bit 56 <-> COM RxPDO-Map Outputs Channel 2/Data Out 7
//     PlcTask Outputs/GVL_SDS.fbSFM_02.stSensSerial.stComOut/D @bit 64 <-> COM RxPDO-Map Outputs Channel 2/Data Out 8
//     PlcTask Outputs/GVL_SDS.fbSFM_02.stSensSerial.stComOut/D @bit 72 <-> COM RxPDO-Map Outputs Channel 2/Data Out 9
//   sample_delivery Instance <-> MAIN (EtherCAT)/Sensirion Flow Meter A Serial 02 (EP6002-0002)
//     PlcTask Inputs/GVL_SDS.fbSFM_03.stSensSerial.stComIn/D <-> COM TxPDO-Map Inputs Channel 1/Data In 0
//     PlcTask Inputs/GVL_SDS.fbSFM_04.stSensSerial.stComIn/D <-> COM TxPDO-Map Inputs Channel 2/Data In 0
//     PlcTask Inputs/GVL_SDS.fbSFM_03.stSensSerial.stComIn/D @bit 8 <-> COM TxPDO-Map Inputs Channel 1/Data In 1
//     PlcTask Inputs/GVL_SDS.fbSFM_03.stSensSerial.stComIn/D @bit 80 <-> COM TxPDO-Map Inputs Channel 1/Data In 10
//     PlcTask Inputs/GVL_SDS.fbSFM_03.stSensSerial.stComIn/D @bit 88 <-> COM TxPDO-Map Inputs Channel 1/Data In 11
//     PlcTask Inputs/GVL_SDS.fbSFM_03.stSensSerial.stComIn/D @bit 96 <-> COM TxPDO-Map Inputs Channel 1/Data In 12
//     PlcTask Inputs/GVL_SDS.fbSFM_03.stSensSerial.stComIn/D @bit 104 <-> COM TxPDO-Map Inputs Channel 1/Data In 13
//     PlcTask Inputs/GVL_SDS.fbSFM_03.stSensSerial.stComIn/D @bit 112 <-> COM TxPDO-Map Inputs Channel 1/Data In 14
//     PlcTask Inputs/GVL_SDS.fbSFM_03.stSensSerial.stComIn/D @bit 120 <-> COM TxPDO-Map Inputs Channel 1/Data In 15
//     PlcTask Inputs/GVL_SDS.fbSFM_03.stSensSerial.stComIn/D @bit 128 <-> COM TxPDO-Map Inputs Channel 1/Data In 16
//     PlcTask Inputs/GVL_SDS.fbSFM_03.stSensSerial.stComIn/D @bit 136 <-> COM TxPDO-Map Inputs Channel 1/Data In 17
//     PlcTask Inputs/GVL_SDS.fbSFM_03.stSensSerial.stComIn/D @bit 144 <-> COM TxPDO-Map Inputs Channel 1/Data In 18
//     PlcTask Inputs/GVL_SDS.fbSFM_03.stSensSerial.stComIn/D @bit 152 <-> COM TxPDO-Map Inputs Channel 1/Data In 19
//     PlcTask Inputs/GVL_SDS.fbSFM_03.stSensSerial.stComIn/D @bit 16 <-> COM TxPDO-Map Inputs Channel 1/Data In 2
//     PlcTask Inputs/GVL_SDS.fbSFM_03.stSensSerial.stComIn/D @bit 160 <-> COM TxPDO-Map Inputs Channel 1/Data In 20
//     PlcTask Inputs/GVL_SDS.fbSFM_03.stSensSerial.stComIn/D @bit 168 <-> COM TxPDO-Map Inputs Channel 1/Data In 21
//     PlcTask Inputs/GVL_SDS.fbSFM_03.stSensSerial.stComIn/D @bit 24 <-> COM TxPDO-Map Inputs Channel 1/Data In 3
//     PlcTask Inputs/GVL_SDS.fbSFM_03.stSensSerial.stComIn/D @bit 32 <-> COM TxPDO-Map Inputs Channel 1/Data In 4
//     PlcTask Inputs/GVL_SDS.fbSFM_03.stSensSerial.stComIn/D @bit 40 <-> COM TxPDO-Map Inputs Channel 1/Data In 5
//     PlcTask Inputs/GVL_SDS.fbSFM_03.stSensSerial.stComIn/D @bit 48 <-> COM TxPDO-Map Inputs Channel 1/Data In 6
//     PlcTask Inputs/GVL_SDS.fbSFM_03.stSensSerial.stComIn/D @bit 56 <-> COM TxPDO-Map Inputs Channel 1/Data In 7
//     PlcTask Inputs/GVL_SDS.fbSFM_03.stSensSerial.stComIn/D @bit 64 <-> COM TxPDO-Map Inputs Channel 1/Data In 8
//     PlcTask Inputs/GVL_SDS.fbSFM_03.stSensSerial.stComIn/D @bit 72 <-> COM TxPDO-Map Inputs Channel 1/Data In 9
//     PlcTask Inputs/GVL_SDS.fbSFM_04.stSensSerial.stComIn/D @bit 8 <-> COM TxPDO-Map Inputs Channel 2/Data In 1
//     PlcTask Inputs/GVL_SDS.fbSFM_04.stSensSerial.stComIn/D @bit 80 <-> COM TxPDO-Map Inputs Channel 2/Data In 10
//     PlcTask Inputs/GVL_SDS.fbSFM_04.stSensSerial.stComIn/D @bit 88 <-> COM TxPDO-Map Inputs Channel 2/Data In 11
//     PlcTask Inputs/GVL_SDS.fbSFM_04.stSensSerial.stComIn/D @bit 96 <-> COM TxPDO-Map Inputs Channel 2/Data In 12
//     PlcTask Inputs/GVL_SDS.fbSFM_04.stSensSerial.stComIn/D @bit 104 <-> COM TxPDO-Map Inputs Channel 2/Data In 13
//     PlcTask Inputs/GVL_SDS.fbSFM_04.stSensSerial.stComIn/D @bit 112 <-> COM TxPDO-Map Inputs Channel 2/Data In 14
//     PlcTask Inputs/GVL_SDS.fbSFM_04.stSensSerial.stComIn/D @bit 120 <-> COM TxPDO-Map Inputs Channel 2/Data In 15
//     PlcTask Inputs/GVL_SDS.fbSFM_04.stSensSerial.stComIn/D @bit 128 <-> COM TxPDO-Map Inputs Channel 2/Data In 16
//     PlcTask Inputs/GVL_SDS.fbSFM_04.stSensSerial.stComIn/D @bit 136 <-> COM TxPDO-Map Inputs Channel 2/Data In 17
//     PlcTask Inputs/GVL_SDS.fbSFM_04.stSensSerial.stComIn/D @bit 144 <-> COM TxPDO-Map Inputs Channel 2/Data In 18
//     PlcTask Inputs/GVL_SDS.fbSFM_04.stSensSerial.stComIn/D @bit 152 <-> COM TxPDO-Map Inputs Channel 2/Data In 19
//     PlcTask Inputs/GVL_SDS.fbSFM_04.stSensSerial.stComIn/D @bit 16 <-> COM TxPDO-Map Inputs Channel 2/Data In 2
//     PlcTask Inputs/GVL_SDS.fbSFM_04.stSensSerial.stComIn/D @bit 160 <-> COM TxPDO-Map Inputs Channel 2/Data In 20
//     PlcTask Inputs/GVL_SDS.fbSFM_04.stSensSerial.stComIn/D @bit 168 <-> COM TxPDO-Map Inputs Channel 2/Data In 21
//     PlcTask Inputs/GVL_SDS.fbSFM_04.stSensSerial.stComIn/D @bit 24 <-> COM TxPDO-Map Inputs Channel 2/Data In 3
//     PlcTask Inputs/GVL_SDS.fbSFM_04.stSensSerial.stComIn/D @bit 32 <-> COM TxPDO-Map Inputs Channel 2/Data In 4
//     PlcTask Inputs/GVL_SDS.fbSFM_04.stSensSerial.stComIn/D @bit 40 <-> COM TxPDO-Map Inputs Channel 2/Data In 5
//     PlcTask Inputs/GVL_SDS.fbSFM_04.stSensSerial.stComIn/D @bit 48 <-> COM TxPDO-Map Inputs Channel 2/Data In 6
//     PlcTask Inputs/GVL_SDS.fbSFM_04.stSensSerial.stComIn/D @bit 56 <-> COM TxPDO-Map Inputs Channel 2/Data In 7
//     PlcTask Inputs/GVL_SDS.fbSFM_04.stSensSerial.stComIn/D @bit 64 <-> COM TxPDO-Map Inputs Channel 2/Data In 8
//     PlcTask Inputs/GVL_SDS.fbSFM_04.stSensSerial.stComIn/D @bit 72 <-> COM TxPDO-Map Inputs Channel 2/Data In 9
//     PlcTask Inputs/GVL_SDS.fbSFM_03.stSensSerial.stComIn/Status <-> COM TxPDO-Map Inputs Channel 1/Status
//     PlcTask Inputs/GVL_SDS.fbSFM_04.stSensSerial.stComIn/Status <-> COM TxPDO-Map Inputs Channel 2/Status
//     PlcTask Outputs/GVL_SDS.fbSFM_03.stSensSerial.stComOut/Ctrl <-> COM RxPDO-Map Outputs Channel 1/Ctrl
//     PlcTask Outputs/GVL_SDS.fbSFM_04.stSensSerial.stComOut/Ctrl <-> COM RxPDO-Map Outputs Channel 2/Ctrl
//     PlcTask Outputs/GVL_SDS.fbSFM_03.stSensSerial.stComOut/D <-> COM RxPDO-Map Outputs Channel 1/Data Out 0
//     PlcTask Outputs/GVL_SDS.fbSFM_04.stSensSerial.stComOut/D <-> COM RxPDO-Map Outputs Channel 2/Data Out 0
//     PlcTask Outputs/GVL_SDS.fbSFM_03.stSensSerial.stComOut/D @bit 8 <-> COM RxPDO-Map Outputs Channel 1/Data Out 1
//     PlcTask Outputs/GVL_SDS.fbSFM_03.stSensSerial.stComOut/D @bit 80 <-> COM RxPDO-Map Outputs Channel 1/Data Out 10
//     PlcTask Outputs/GVL_SDS.fbSFM_03.stSensSerial.stComOut/D @bit 88 <-> COM RxPDO-Map Outputs Channel 1/Data Out 11
//     PlcTask Outputs/GVL_SDS.fbSFM_03.stSensSerial.stComOut/D @bit 96 <-> COM RxPDO-Map Outputs Channel 1/Data Out 12
//     PlcTask Outputs/GVL_SDS.fbSFM_03.stSensSerial.stComOut/D @bit 104 <-> COM RxPDO-Map Outputs Channel 1/Data Out 13
//     PlcTask Outputs/GVL_SDS.fbSFM_03.stSensSerial.stComOut/D @bit 112 <-> COM RxPDO-Map Outputs Channel 1/Data Out 14
//     PlcTask Outputs/GVL_SDS.fbSFM_03.stSensSerial.stComOut/D @bit 120 <-> COM RxPDO-Map Outputs Channel 1/Data Out 15
//     PlcTask Outputs/GVL_SDS.fbSFM_03.stSensSerial.stComOut/D @bit 128 <-> COM RxPDO-Map Outputs Channel 1/Data Out 16
//     PlcTask Outputs/GVL_SDS.fbSFM_03.stSensSerial.stComOut/D @bit 136 <-> COM RxPDO-Map Outputs Channel 1/Data Out 17
//     PlcTask Outputs/GVL_SDS.fbSFM_03.stSensSerial.stComOut/D @bit 144 <-> COM RxPDO-Map Outputs Channel 1/Data Out 18
//     PlcTask Outputs/GVL_SDS.fbSFM_03.stSensSerial.stComOut/D @bit 152 <-> COM RxPDO-Map Outputs Channel 1/Data Out 19
//     PlcTask Outputs/GVL_SDS.fbSFM_03.stSensSerial.stComOut/D @bit 16 <-> COM RxPDO-Map Outputs Channel 1/Data Out 2
//     PlcTask Outputs/GVL_SDS.fbSFM_03.stSensSerial.stComOut/D @bit 160 <-> COM RxPDO-Map Outputs Channel 1/Data Out 20
//     PlcTask Outputs/GVL_SDS.fbSFM_03.stSensSerial.stComOut/D @bit 168 <-> COM RxPDO-Map Outputs Channel 1/Data Out 21
//     PlcTask Outputs/GVL_SDS.fbSFM_03.stSensSerial.stComOut/D @bit 24 <-> COM RxPDO-Map Outputs Channel 1/Data Out 3
//     PlcTask Outputs/GVL_SDS.fbSFM_03.stSensSerial.stComOut/D @bit 32 <-> COM RxPDO-Map Outputs Channel 1/Data Out 4
//     PlcTask Outputs/GVL_SDS.fbSFM_03.stSensSerial.stComOut/D @bit 40 <-> COM RxPDO-Map Outputs Channel 1/Data Out 5
//     PlcTask Outputs/GVL_SDS.fbSFM_03.stSensSerial.stComOut/D @bit 48 <-> COM RxPDO-Map Outputs Channel 1/Data Out 6
//     PlcTask Outputs/GVL_SDS.fbSFM_03.stSensSerial.stComOut/D @bit 56 <-> COM RxPDO-Map Outputs Channel 1/Data Out 7
//     PlcTask Outputs/GVL_SDS.fbSFM_03.stSensSerial.stComOut/D @bit 64 <-> COM RxPDO-Map Outputs Channel 1/Data Out 8
//     PlcTask Outputs/GVL_SDS.fbSFM_03.stSensSerial.stComOut/D @bit 72 <-> COM RxPDO-Map Outputs Channel 1/Data Out 9
//     PlcTask Outputs/GVL_SDS.fbSFM_04.stSensSerial.stComOut/D @bit 8 <-> COM RxPDO-Map Outputs Channel 2/Data Out 1
//     PlcTask Outputs/GVL_SDS.fbSFM_04.stSensSerial.stComOut/D @bit 80 <-> COM RxPDO-Map Outputs Channel 2/Data Out 10
//     PlcTask Outputs/GVL_SDS.fbSFM_04.stSensSerial.stComOut/D @bit 88 <-> COM RxPDO-Map Outputs Channel 2/Data Out 11
//     PlcTask Outputs/GVL_SDS.fbSFM_04.stSensSerial.stComOut/D @bit 96 <-> COM RxPDO-Map Outputs Channel 2/Data Out 12
//     PlcTask Outputs/GVL_SDS.fbSFM_04.stSensSerial.stComOut/D @bit 104 <-> COM RxPDO-Map Outputs Channel 2/Data Out 13
//     PlcTask Outputs/GVL_SDS.fbSFM_04.stSensSerial.stComOut/D @bit 112 <-> COM RxPDO-Map Outputs Channel 2/Data Out 14
//     PlcTask Outputs/GVL_SDS.fbSFM_04.stSensSerial.stComOut/D @bit 120 <-> COM RxPDO-Map Outputs Channel 2/Data Out 15
//     PlcTask Outputs/GVL_SDS.fbSFM_04.stSensSerial.stComOut/D @bit 128 <-> COM RxPDO-Map Outputs Channel 2/Data Out 16
//     PlcTask Outputs/GVL_SDS.fbSFM_04.stSensSerial.stComOut/D @bit 136 <-> COM RxPDO-Map Outputs Channel 2/Data Out 17
//     PlcTask Outputs/GVL_SDS.fbSFM_04.stSensSerial.stComOut/D @bit 144 <-> COM RxPDO-Map Outputs Channel 2/Data Out 18
//     PlcTask Outputs/GVL_SDS.fbSFM_04.stSensSerial.stComOut/D @bit 152 <-> COM RxPDO-Map Outputs Channel 2/Data Out 19
//     PlcTask Outputs/GVL_SDS.fbSFM_04.stSensSerial.stComOut/D @bit 16 <-> COM RxPDO-Map Outputs Channel 2/Data Out 2
//     PlcTask Outputs/GVL_SDS.fbSFM_04.stSensSerial.stComOut/D @bit 160 <-> COM RxPDO-Map Outputs Channel 2/Data Out 20
//     PlcTask Outputs/GVL_SDS.fbSFM_04.stSensSerial.stComOut/D @bit 168 <-> COM RxPDO-Map Outputs Channel 2/Data Out 21
//     PlcTask Outputs/GVL_SDS.fbSFM_04.stSensSerial.stComOut/D @bit 24 <-> COM RxPDO-Map Outputs Channel 2/Data Out 3
//     PlcTask Outputs/GVL_SDS.fbSFM_04.stSensSerial.stComOut/D @bit 32 <-> COM RxPDO-Map Outputs Channel 2/Data Out 4
//     PlcTask Outputs/GVL_SDS.fbSFM_04.stSensSerial.stComOut/D @bit 40 <-> COM RxPDO-Map Outputs Channel 2/Data Out 5
//     PlcTask Outputs/GVL_SDS.fbSFM_04.stSensSerial.stComOut/D @bit 48 <-> COM RxPDO-Map Outputs Channel 2/Data Out 6
//     PlcTask Outputs/GVL_SDS.fbSFM_04.stSensSerial.stComOut/D @bit 56 <-> COM RxPDO-Map Outputs Channel 2/Data Out 7
//     PlcTask Outputs/GVL_SDS.fbSFM_04.stSensSerial.stComOut/D @bit 64 <-> COM RxPDO-Map Outputs Channel 2/Data Out 8
//     PlcTask Outputs/GVL_SDS.fbSFM_04.stSensSerial.stComOut/D @bit 72 <-> COM RxPDO-Map Outputs Channel 2/Data Out 9
//   sample_delivery Instance <-> MAIN (EtherCAT)/Solenoid Pair A Digital IO (EP2338-0001)
//     PlcTask Outputs/GVL_SDS.PURGE_VRC_01_CTL <-> Channel 12/Output
//     PlcTask Outputs/GVL_SDS.PURGE_VRC_02_CTL <-> Channel 13/Output
//     PlcTask Outputs/GVL_SDS.SolenoidPairA.q_xDO1 <-> Channel 9/Output
//     PlcTask Outputs/GVL_SDS.SolenoidPairA.q_xDO2 <-> Channel 10/Output
//   sample_delivery Instance <-> MAIN (EtherCAT)/WALL-RCC (EP2338-0001)
//     PlcTask Inputs/GVL_Recirculation.RCC_VRC_01.i_xOpnLS <-> Channel 1/Input
//     PlcTask Inputs/GVL_Recirculation.RCC_VRC_02.i_xOpnLS <-> Channel 2/Input
//     PlcTask Inputs/GVL_Recirculation.RCC_VRC_03.i_xOpnLS <-> Channel 3/Input
//     PlcTask Inputs/GVL_Recirculation.RCC_VRC_04.i_xOpnLS <-> Channel 4/Input
//     PlcTask Outputs/GVL_Recirculation.RCC_VRC_01.q_xOPN_DO <-> Channel 9/Output
//     PlcTask Outputs/GVL_Recirculation.RCC_VRC_02.q_xOPN_DO <-> Channel 10/Output
//     PlcTask Outputs/GVL_Recirculation.RCC_VRC_03.q_xOPN_DO <-> Channel 11/Output
//     PlcTask Outputs/GVL_Recirculation.RCC_VRC_04.q_xOPN_DO <-> Channel 12/Output
//   sample_delivery Instance <-> MAIN (EtherCAT)/WALL-RCC-PCM (EP4374-0002)
//     PlcTask Inputs/PRG_WALL_RCC.PCM_RCC.stPropAir1.i_iPressRB <-> AI Inputs Channel 1/Value
//     PlcTask Inputs/PRG_WALL_RCC.PCM_RCC.stPropAir2.i_iPressRB <-> AI Inputs Channel 2/Value
//     PlcTask Outputs/PRG_WALL_RCC.PCM_RCC.stPropAir1.q_iPressCt <-> AO Outputs Channel 3/Analog output
//     PlcTask Outputs/PRG_WALL_RCC.PCM_RCC.stPropAir2.q_iPressCt <-> AO Outputs Channel 4/Analog output

// ---- GVLs/GVL_RCC.TcGVL
VAR_GLOBAL
{attribute 'pytmc' :=' pv: XCS:RCC:VRC:01 '}
{attribute 'TcLinkTo' := 	'.i_xOpnLS	:=	TIIB[RCC (EP2338-0001)]^Channel 1^Input;
                             .q_xOPN_DO	:=	TIIB[RCC (EP2338-0001)]^Channel 9^Output'}
 RCC_VRC_01 : FB_VRC_NC_OPNLS;

{attribute 'pytmc' :=' pv: XCS:RCC:VRC:02 '}
{attribute 'TcLinkTo' := 	'.i_xOpnLS	:=	TIIB[RCC (EP2338-0001)]^Channel 2^Input;
                             .q_xOPN_DO	:=	TIIB[RCC (EP2338-0001)]^Channel 10^Output'}
 RCC_VRC_02 : FB_VRC_NC_OPNLS;
{attribute 'pytmc' :=' pv: XCS:RCC:VRC:03 '}
{attribute 'TcLinkTo' := 	'.i_xOpnLS	:=	TIIB[RCC (EP2338-0001)]^Channel 3^Input;
                             .q_xOPN_DO	:=	TIIB[RCC (EP2338-0001)]^Channel 11^Output'}
 RCC_VRC_03 : FB_VRC_NC_OPNLS;
{attribute 'pytmc' :=' pv: XCS:RCC:VRC:04 '}
{attribute 'TcLinkTo' := 	'.i_xOpnLS	:=	TIIB[RCC (EP2338-0001)]^Channel 4^Input;
                             .q_xOPN_DO	:=	TIIB[RCC (EP2338-0001)]^Channel 12^Output'}
 RCC_VRC_04 : FB_VRC_NC_OPNLS;

// RCC PUMP
{attribute 'pytmc' :=' pv: XCS:RCC:VRC:05 '}
{attribute 'TcLinkTo' := 	'.i_xOpnLS	:=	TIIB[RCC (EP2338-0001)]^Channel 5^Input;
                             .q_xOPN_DO	:=	TIIB[RCC (EP2338-0001)]^Channel 13^Output'}
 RCC_VRC_05 : FB_VRC_NC_OPNLS;

{attribute 'pytmc' :=' pv: XCS:RCC:VRC:06 '}
{attribute 'TcLinkTo' := 	'.i_xOpnLS	:=	TIIB[RCC (EP2338-0001)]^Channel 6^Input;
                             .q_xOPN_DO	:=	TIIB[RCC (EP2338-0001)]^Channel 14^Output'}
 RCC_VRC_06 : FB_VRC_NC_OPNLS;
{attribute 'pytmc' :=' pv: XCS:RCC:VRC:07 '}
{attribute 'TcLinkTo' := 	'.i_xOpnLS	:=	TIIB[RCC (EP2338-0001)]^Channel 7^Input;
                             .q_xOPN_DO	:=	TIIB[RCC (EP2338-0001)]^Channel 15^Output'}
 RCC_VRC_07 : FB_VRC_NC_OPNLS;
{attribute 'pytmc' :=' pv: XCS:RCC:VRC:08 '}
{attribute 'TcLinkTo' := 	'.i_xOpnLS	:=	TIIB[RCC (EP2338-0001)]^Channel 8^Input;
                             .q_xOPN_DO	:=	TIIB[RCC (EP2338-0001)]^Channel 16^Output'}
 RCC_VRC_08 : FB_VRC_NC_OPNLS;

END_VAR

// ---- GVLs/GVL_SDS.TcGVL
VAR_GLOBAL

// TODO: FIX Linking for Devices will be deployed
//  Working: Bronkhorst MFM B
{attribute 'pytmc' := 'pv: XCS:SDS:SEL:A'}
{attribute 'TcLinkTo' := '.stSensSerial.stComIn.Status := TIIB[M3 Selector A Serial IO (EP6002-0002)]^COM TxPDO-Map Inputs Channel 1^Status;
                          .stViciSerial.stComIn.Status := TIIB[M3 Selector A Serial IO (EP6002-0002)]^COM TxPDO-Map Inputs Channel 2^Status;
                          .stSensSerial.stComOut.Ctrl := TIID^MAIN (EtherCAT)^M3 Selector A Serial IO (EP6002-0002)^COM RxPDO-Map Outputs Channel 1^Ctrl;
                          .stViciSerial.stComOut.Ctrl := TIID^MAIN (EtherCAT)^M3 Selector A Serial IO (EP6002-0002)^COM RxPDO-Map Outputs Channel 2^Ctrl;
                          .stShaker01.q_xPwrDO := TIIB[M3 Selector A Digital IO (EP2338-1001)]^Channel 9^Output;
                          .stShaker02.q_xPwrDO := TIIB[M3 Selector A Digital IO (EP2338-1001)]^Channel 10^Output;
                          .stShaker03.q_xPwrDO := TIIB[M3 Selector A Digital IO (EP2338-1001)]^Channel 11^Output;
                          .stShaker04.q_xPwrDO := TIIB[M3 Selector A Digital IO (EP2338-1001)]^Channel 12^Output;
                          .stBaseIO.i_SyncUnitWC := TIID^MAIN (EtherCAT)^M3 Selector A (EP1111)^WcState^WcState;
                          .
'}
M3SelectorA : FB_SelectorM3;

{attribute 'pytmc' := 'pv: XCS:SDS:SEL:B'}
{attribute 'TcLinkTo' := '.stSensSerial.stComIn.Status := TIIB[M3 Selector B Serial IO (EP6002-0002)]^COM TxPDO-Map Inputs Channel 1^Status;
                          .stViciSerial.stComIn.Status := TIIB[M3 Selector B Serial IO (EP6002-0002)]^COM TxPDO-Map Inputs Channel 2^Status;
                          .stSensSerial.stComOut.Ctrl := TIID^MAIN (EtherCAT)^M3 Selector B Serial IO (EP6002-0002)^COM RxPDO-Map Outputs Channel 1^Ctrl;
                          .stViciSerial.stComOut.Ctrl := TIID^MAIN (EtherCAT)^M3 Selector B Serial IO (EP6002-0002)^COM RxPDO-Map Outputs Channel 2^Ctrl;
                          .stShaker01.q_xPwrDO := TIIB[M3 Selector B Digital IO (EP2338-1001)]^Channel 9^Output;
                          .stShaker02.q_xPwrDO := TIIB[M3 Selector B Digital IO (EP2338-1001)]^Channel 10^Output;
                          .stShaker03.q_xPwrDO := TIIB[M3 Selector B Digital IO (EP2338-1001)]^Channel 11^Output;
                          .stShaker04.q_xPwrDO := TIIB[M3 Selector B Digital IO (EP2338-1001)]^Channel 12^Output;
                          .stBaseIO.i_SyncUnitWC := TIID^MAIN (EtherCAT)^M3 Selector B (EP1111)^WcState^WcState
'}
M3SelectorB : FB_SelectorM3;

{attribute 'pytmc' := 'pv: XCS:SDS:SEL:C'}
{attribute 'TcLinkTo' := '.stSensSerial.stComIn.Status := TIIB[M3 Selector C Serial IO (EP6002-0002)]^COM TxPDO-Map Inputs Channel 1^Status;
                          .stViciSerial.stComIn.Status := TIIB[M3 Selector C Serial IO (EP6002-0002)]^COM TxPDO-Map Inputs Channel 2^Status;
                          .stSensSerial.stComOut.Ctrl := TIID^MAIN (EtherCAT)^M3 Selector C Serial IO (EP6002-0002)^COM RxPDO-Map Outputs Channel 1^Ctrl;
                          .stViciSerial.stComOut.Ctrl := TIID^MAIN (EtherCAT)^M3 Selector C Serial IO (EP6002-0002)^COM RxPDO-Map Outputs Channel 2^Ctrl;
                          .stShaker01.q_xPwrDO := TIIB[M3 Selector C Digital IO (EP2338-1001)]^Channel 9^Output;
                          .stShaker02.q_xPwrDO := TIIB[M3 Selector C Digital IO (EP2338-1001)]^Channel 10^Output;
                          .stShaker03.q_xPwrDO := TIIB[M3 Selector C Digital IO (EP2338-1001)]^Channel 11^Output;
                          .stShaker04.q_xPwrDO := TIIB[M3 Selector C Digital IO (EP2338-1001)]^Channel 12^Output;
                          .stBaseIO.i_SyncUnitWC := TIID^MAIN (EtherCAT)^M3 Selector C (EP1111)^WcState^WcState
'}
M3SelectorC : FB_SelectorM3;

{attribute 'pytmc' := 'pv: XCS:SDS:SEL:D'}
{attribute 'TcLinkTo' := '.stSensSerial.stComIn.Status := TIIB[M3 Selector D Serial IO (EP6002-0002)]^COM TxPDO-Map Inputs Channel 1^Status;
                          .stViciSerial.stComIn.Status := TIIB[M3 Selector D Serial IO (EP6002-0002)]^COM TxPDO-Map Inputs Channel 2^Status;
                          .stSensSerial.stComOut.Ctrl := TIID^MAIN (EtherCAT)^M3 Selector D Serial IO (EP6002-0002)^COM RxPDO-Map Outputs Channel 1^Ctrl;
                          .stViciSerial.stComOut.Ctrl := TIID^MAIN (EtherCAT)^M3 Selector D Serial IO (EP6002-0002)^COM RxPDO-Map Outputs Channel 2^Ctrl;
                          .stShaker01.q_xPwrDO := TIIB[M3 Selector D Digital IO (EP2338-1001)]^Channel 9^Output;
                          .stShaker02.q_xPwrDO := TIIB[M3 Selector D Digital IO (EP2338-1001)]^Channel 10^Output;
                          .stShaker03.q_xPwrDO := TIIB[M3 Selector D Digital IO (EP2338-1001)]^Channel 11^Output;
                          .stShaker04.q_xPwrDO := TIIB[M3 Selector D Digital IO (EP2338-1001)]^Channel 12^Output;
                          .stBaseIO.i_SyncUnitWC := TIID^MAIN (EtherCAT)^M3 Selector D (EP1111)^WcState^WcState
'}
M3SelectorD : FB_SelectorM3;

{attribute 'pytmc' := 'pv: XCS:SDS:PCM:A'}
{attribute 'TcLinkTo' := '.stPropAir1.i_iPressRB 		:= TIIB[PCM A (EP4374-0002)]^AI Inputs Channel 1^Value;
                          .stPropAir2.i_iPressRB 		:= TIIB[PCM A (EP4374-0002)]^AI Inputs Channel 2^Value;
                          .stPropAir1.q_iPressCt 		:= TIIB[PCM A (EP4374-0002)]^AO Outputs Channel 3^Analog output;
                          .stPropAir2.q_iPressCt 		:= TIIB[PCM A (EP4374-0002)]^AO Outputs Channel 4^Analog output;
                          .stSerial1.stComIn.Status 	:= TIIB[PCM A (EP6002-0002)]^COM TxPDO-Map Inputs Channel 1^Status;
                          .stSerial2.stComIn.Status 	:= TIIB[PCM A (EP6002-0002)]^COM TxPDO-Map Inputs Channel 2^Status;
                          .stSerial1.stComOut.Ctrl 		:= TIIB[PCM A (EP6002-0002)]^COM RxPDO-Map Outputs Channel 1^Ctrl;
                          .stSerial2.stComOut.Ctrl 		:= TIIB[PCM A (EP6002-0002)]^COM RxPDO-Map Outputs Channel 2^Ctrl;
                          .stBaseIO.i_SyncUnitWC 		:= TIIB[PCM A (EP1111)]^WcState^WcState;

                          .stSerial1.stComIn.D[0]  		:= TIIB[PCM A (EP6002-0002)]^COM TxPDO-Map Inputs Channel 1^Data In 0;
                          .stSerial1.stComIn.D[1]  		:= TIIB[PCM A (EP6002-0002)]^COM TxPDO-Map Inputs Channel 1^Data In 1;
                          .stSerial1.stComIn.D[2]  		:= TIIB[PCM A (EP6002-0002)]^COM TxPDO-Map Inputs Channel 1^Data In 2;
                          .stSerial1.stComIn.D[3]  		:= TIIB[PCM A (EP6002-0002)]^COM TxPDO-Map Inputs Channel 1^Data In 3;
                          .stSerial1.stComIn.D[4]  		:= TIIB[PCM A (EP6002-0002)]^COM TxPDO-Map Inputs Channel 1^Data In 4;
                          .stSerial1.stComIn.D[5]  		:= TIIB[PCM A (EP6002-0002)]^COM TxPDO-Map Inputs Channel 1^Data In 5;
                          .stSerial1.stComIn.D[6]  		:= TIIB[PCM A (EP6002-0002)]^COM TxPDO-Map Inputs Channel 1^Data In 6;
                          .stSerial1.stComIn.D[7]  		:= TIIB[PCM A (EP6002-0002)]^COM TxPDO-Map Inputs Channel 1^Data In 7;
                          .stSerial1.stComIn.D[8]  		:= TIIB[PCM A (EP6002-0002)]^COM TxPDO-Map Inputs Channel 1^Data In 8;
                          .stSerial1.stComIn.D[9]  		:= TIIB[PCM A (EP6002-0002)]^COM TxPDO-Map Inputs Channel 1^Data In 9;
                          .stSerial1.stComIn.D[10]  	:= TIIB[PCM A (EP6002-0002)]^COM TxPDO-Map Inputs Channel 1^Data In 10;
                          .stSerial1.stComIn.D[11]  	:= TIIB[PCM A (EP6002-0002)]^COM TxPDO-Map Inputs Channel 1^Data In 11;
                          .stSerial1.stComIn.D[12]  	:= TIIB[PCM A (EP6002-0002)]^COM TxPDO-Map Inputs Channel 1^Data In 12;
                          .stSerial1.stComIn.D[13]  	:= TIIB[PCM A (EP6002-0002)]^COM TxPDO-Map Inputs Channel 1^Data In 13;
                          .stSerial1.stComIn.D[14]  	:= TIIB[PCM A (EP6002-0002)]^COM TxPDO-Map Inputs Channel 1^Data In 14;
                          .stSerial1.stComIn.D[15]  	:= TIIB[PCM A (EP6002-0002)]^COM TxPDO-Map Inputs Channel 1^Data In 15;
                          .stSerial1.stComIn.D[16]  	:= TIIB[PCM A (EP6002-0002)]^COM TxPDO-Map Inputs Channel 1^Data In 16;
                          .stSerial1.stComIn.D[17]  	:= TIIB[PCM A (EP6002-0002)]^COM TxPDO-Map Inputs Channel 1^Data In 17;
                          .stSerial1.stComIn.D[18]  	:= TIIB[PCM A (EP6002-0002)]^COM TxPDO-Map Inputs Channel 1^Data In 18;
                          .stSerial1.stComIn.D[19]  	:= TIIB[PCM A (EP6002-0002)]^COM TxPDO-Map Inputs Channel 1^Data In 19;
                          .stSerial1.stComIn.D[20]  	:= TIIB[PCM A (EP6002-0002)]^COM TxPDO-Map Inputs Channel 1^Data In 20;
                          .stSerial1.stComIn.D[21]  	:= TIIB[PCM A (EP6002-0002)]^COM TxPDO-Map Inputs Channel 1^Data In 21;

                          .stSerial2.stComIn.D[0]  		:= TIIB[PCM A (EP6002-0002)]^COM TxPDO-Map Inputs Channel 2^Data In 0;
                          .stSerial2.stComIn.D[1]  		:= TIIB[PCM A (EP6002-0002)]^COM TxPDO-Map Inputs Channel 2^Data In 1;
                          .stSerial2.stComIn.D[2]  		:= TIIB[PCM A (EP6002-0002)]^COM TxPDO-Map Inputs Channel 2^Data In 2;
                          .stSerial2.stComIn.D[3]  		:= TIIB[PCM A (EP6002-0002)]^COM TxPDO-Map Inputs Channel 2^Data In 3;
                          .stSerial2.stComIn.D[4]  		:= TIIB[PCM A (EP6002-0002)]^COM TxPDO-Map Inputs Channel 2^Data In 4;
                          .stSerial2.stComIn.D[5]  		:= TIIB[PCM A (EP6002-0002)]^COM TxPDO-Map Inputs Channel 2^Data In 5;
                          .stSerial2.stComIn.D[6]  		:= TIIB[PCM A (EP6002-0002)]^COM TxPDO-Map Inputs Channel 2^Data In 6;
                          .stSerial2.stComIn.D[7]  		:= TIIB[PCM A (EP6002-0002)]^COM TxPDO-Map Inputs Channel 2^Data In 7;
                          .stSerial2.stComIn.D[8]  		:= TIIB[PCM A (EP6002-0002)]^COM TxPDO-Map Inputs Channel 2^Data In 8;
                          .stSerial2.stComIn.D[9]  		:= TIIB[PCM A (EP6002-0002)]^COM TxPDO-Map Inputs Channel 2^Data In 9;
                          .stSerial2.stComIn.D[10]  	:= TIIB[PCM A (EP6002-0002)]^COM TxPDO-Map Inputs Channel 2^Data In 10;
                          .stSerial2.stComIn.D[11]  	:= TIIB[PCM A (EP6002-0002)]^COM TxPDO-Map Inputs Channel 2^Data In 11;
                          .stSerial2.stComIn.D[12]  	:= TIIB[PCM A (EP6002-0002)]^COM TxPDO-Map Inputs Channel 2^Data In 12;
                          .stSerial2.stComIn.D[13]  	:= TIIB[PCM A (EP6002-0002)]^COM TxPDO-Map Inputs Channel 2^Data In 13;
                          .stSerial2.stComIn.D[14]  	:= TIIB[PCM A (EP6002-0002)]^COM TxPDO-Map Inputs Channel 2^Data In 14;
                          .stSerial2.stComIn.D[15]  	:= TIIB[PCM A (EP6002-0002)]^COM TxPDO-Map Inputs Channel 2^Data In 15;
                          .stSerial2.stComIn.D[16]  	:= TIIB[PCM A (EP6002-0002)]^COM TxPDO-Map Inputs Channel 2^Data In 16;
                          .stSerial2.stComIn.D[17]  	:= TIIB[PCM A (EP6002-0002)]^COM TxPDO-Map Inputs Channel 2^Data In 17;
                          .stSerial2.stComIn.D[18]  	:= TIIB[PCM A (EP6002-0002)]^COM TxPDO-Map Inputs Channel 2^Data In 18;
                          .stSerial2.stComIn.D[19]  	:= TIIB[PCM A (EP6002-0002)]^COM TxPDO-Map Inputs Channel 2^Data In 19;
                          .stSerial2.stComIn.D[20]  	:= TIIB[PCM A (EP6002-0002)]^COM TxPDO-Map Inputs Channel 2^Data In 20;
                          .stSerial2.stComIn.D[21]  	:= TIIB[PCM A (EP6002-0002)]^COM TxPDO-Map Inputs Channel 2^Data In 21;

